ELSIF ref.driveTripOK THEN
    IF ref.driveRelease THEN
        driveStatus.color.fg := COLORS.BLACK;
        driveStatus.color.bg := COLORS.GREEN;
        IF ref.driveMinFrequency THEN
            _formatString(sFormat := '%.1f Hz',  arg1 := F_LREAL(ref.frequencyMeasurement.average.hertz.value), sOut => driveStatus.text);
        ELSE
            _formatString(sFormat := '%.1f Hz (LOW)',  arg1 := F_LREAL(ref.frequencyMeasurement.average.hertz.value), sOut => driveStatus.text);
		END_IF
    ELSE
        driveStatus.color.fg := COLORS.BLACK;
        driveStatus.color.bg := COLORS.GRAY;
        driveStatus.text := 'Not released';
	END_IF
ELSE
        driveStatus.color.fg := COLORS.WHITE;
        driveStatus.color.bg := COLORS.RED;
        driveStatus.text := 'TRIPPED';
END_IF

// update the pressureStatus
pressureStatus(color := HealthToColor(ref.pressureMeasurement.statuses.healthStatus));
_formatString(sFormat := '%.1f Bar',  arg1 := F_LREAL(ref.pressureMeasurement.average.bar.value), sOut => pressureStatus.text);

END_FUNCTION_BLOCK

// ---- MTCS/Hydraulics/Widgets/HydraulicsIOWidget.TcPOU
FUNCTION_BLOCK HydraulicsIOWidget
VAR_INPUT
END_VAR
VAR_OUTPUT
END_VAR
VAR
	actualStatus : StatusWidget;
	pumpsGroup : HydraulicsPumpsGroupIOWidget;
    hydraulicsAndSafety : SafetyHydraulicsAndSafetyIOWidget;
END_VAR
VAR_IN_OUT
	ref : HydraulicsIO;
	ref_safetyIO : SafetyIO;
END_VAR

actualStatus(text  := ref.actualStatus,
             color := HealthToColor(ref.statuses.healthStatus));

pumpsGroup(ref := ref.parts.pumpsGroup);
hydraulicsAndSafety(ref := ref_safetyIO.parts.hydraulicsAndSafety);

END_FUNCTION_BLOCK

// ---- MTCS/Hydraulics/Widgets/HydraulicsPumpsGroupIOWidget.TcPOU
FUNCTION_BLOCK HydraulicsPumpsGroupIOWidget
VAR_INPUT
END_VAR
VAR_OUTPUT
END_VAR
VAR
	actualStatus : StatusWidget;
    
	COU : EtherCatDeviceWidget;
	DI1 : EtherCatDeviceWidget;
	SI1 : EtherCatDeviceWidget;
	SI2 : EtherCatDeviceWidget;
	SI3 : EtherCatDeviceWidget;
	DI2 : EtherCatDeviceWidget;
END_VAR
VAR_IN_OUT
	ref : HydraulicsPumpsGroupIO;
END_VAR

actualStatus(text  := ref.actualStatus,
             color := HealthToColor(ref.statuses.healthStatus));

COU(device := ref.parts.COU);
DI1(device := ref.parts.DI1);
SI1(device := ref.parts.SI1);
SI2(device := ref.parts.SI2);
SI3(device := ref.parts.SI3);
DI2(device := ref.parts.DI2);

END_FUNCTION_BLOCK

// ---- MTCS/Hydraulics/Widgets/HydraulicsWidget.TcPOU
FUNCTION_BLOCK HydraulicsWidget
VAR_INPUT
END_VAR
VAR_OUTPUT
    configManager : ConfigManagerWidget;
	initializationStatus : InitializationStatusWidget;
	actualStatus : StatusWidget;
	pumpsStatus : StatusWidget;
    name : STRING := 'Hydraulics';
    
END_VAR
VAR_IN_OUT
	ref : Hydraulics;
    ref_safetyIO : SafetyIO;
END_VAR
VAR
    io : HydraulicsIOWidget;
    
    button_initialize : InitializeButtonWidget;
    button_operating  : OperatingButtonWidget;
    button_locking    : LockingButtonWidget;
    
    activeTab       : HydraulicsTabs := HydraulicsTabs.OVERVIEW;
    button_overview : SubSystemButtonWidget('Overview'      , HydraulicsTabs.OVERVIEW);
    button_technical: SubSystemButtonWidget('Technical'     , HydraulicsTabs.TECHNICAL);
    button_io       : SubSystemButtonWidget('I/O'           , HydraulicsTabs.IO);
    button_config   : SubSystemButtonWidget('Config'        , HydraulicsTabs.CONFIG);
    
    top             : HydraulicsSideWidget;
    bottom          : HydraulicsSideWidget;
    
	bearingTemperatureStatus : StatusWidget;
    
    _formatString : FB_FormatString;
    activeConfigTab : INT;
    
    bearingTemperature  : MeasurementWidget('Bearing temperature', '%.2f °C');
    topFrequencyMeasurement  : MeasurementWidget('Top drive output frequency', '%.2f Hz');
    topPressureMeasurement  : MeasurementWidget('Top pressure', '%.2f Bar');
    bottomFrequencyMeasurement  : MeasurementWidget('Bottom drive output frequency', '%.2f Hz');
    bottomPressureMeasurement  : MeasurementWidget('Bottom pressure', '%.2f Bar');
    
    circulationStatus : StatusWidget;
    circulationPumpRelay : SimpleRelayWidget;
    pumpsPowerRelay : SimpleRelayWidget;
END_VAR

initializationStatus(status := ref.statuses.initializationStatus);
configManager(mgr := ref.parts.configManager);

actualStatus(text  := ref.actualStatus,
             color := SystemToColor(healthStatus := ref.statuses.healthStatus,
                                    busyStatus   := ref.statuses.busyStatus,
                                    initializationStatus := ref.statuses.initializationStatus,
                                    operatingStatus := ref.statuses.operatingStatus));

pumpsStatus(text  := ref.pumpsStatus, color := actualStatus.color);
                                    
io(ref := ref.parts.io, ref_safetyIO := ref_safetyIO);

button_initialize(status := ref.statuses.initializationStatus, process := ref.processes.initialize);
button_operating(status := ref.statuses.operatingStatus, process := ref.processes.changeOperatingState);
button_locking(status := ref.statuses.initializationStatus, lock := ref.processes.lock, unlock := ref.processes.unlock);

button_overview(    color := actualStatus.color                 , activeTab := activeTab);
button_technical(   color := actualStatus.color                 , activeTab := activeTab);
button_io(          color := io.actualStatus.color              , activeTab := activeTab);
button_config(      color := configManager.actualStatus.color   , activeTab := activeTab);

top(ref := ref.parts.top, powered := ref.parts.pumpsPowerRelay.digitalOutput);
bottom(ref := ref.parts.bottom, powered := ref.parts.pumpsPowerRelay.digitalOutput);

bearingTemperatureStatus(color := HealthToColor(ref.bearingTemperature.statuses.healthStatus));
_formatString(sFormat := '%.1f °C',  arg1 := F_LREAL(ref.bearingTemperature.average.celsius.value), sOut => bearingTemperatureStatus.text);


bearingTemperature(value        := ref.bearingTemperature.average.celsius.value, 
                   actualStatus := ref.bearingTemperature.actualStatus, 
                   healthStatus := ref.bearingTemperature.statuses.healthStatus);
topFrequencyMeasurement(value        := ref.parts.top.frequencyMeasurement.average.hertz.value, 
                        actualStatus := ref.parts.top.frequencyMeasurement.actualStatus, 
                        healthStatus := ref.parts.top.frequencyMeasurement.statuses.healthStatus);
bottomFrequencyMeasurement( value        := ref.parts.bottom.frequencyMeasurement.average.hertz.value, 
                            actualStatus := ref.parts.bottom.frequencyMeasurement.actualStatus, 
                            healthStatus := ref.parts.bottom.frequencyMeasurement.statuses.healthStatus);
topPressureMeasurement(value        := ref.parts.top.pressureMeasurement.average.bar.value, 
                        actualStatus := ref.parts.top.pressureMeasurement.actualStatus, 
                        healthStatus := ref.parts.top.pressureMeasurement.statuses.healthStatus);
bottomPressureMeasurement(value        := ref.parts.bottom.pressureMeasurement.average.bar.value, 
                          actualStatus := ref.parts.bottom.pressureMeasurement.actualStatus, 
                          healthStatus := ref.parts.bottom.pressureMeasurement.statuses.healthStatus);

IF ref.parts.circulationPumpRelay.digitalOutput THEN
    circulationStatus.text := 'ON';
    circulationStatus.color.fg := Colors.BLACK;
    circulationStatus.color.bg := Colors.GREEN;
ELSE
    circulationStatus.text := 'OFF';
    circulationStatus.color.fg := Colors.BLACK;
    circulationStatus.color.bg := Colors.GRAY;
END_IF

circulationPumpRelay(ref := ref.parts.circulationPumpRelay);
pumpsPowerRelay(ref := ref.parts.pumpsPowerRelay);

END_FUNCTION_BLOCK

// ---- MTCS/M1/StateMachines/M1AxialSupport.TcPOU
FUNCTION_BLOCK M1AxialSupport EXTENDS SM_M1AxialSupport
VAR_INPUT
END_VAR
VAR_OUTPUT
END_VAR
VAR
    _unlimitedAutoForceSetpointDaN : LREAL;
    
	_executeController : BOOL;
    _ctrl_pi : FB_CTRL_PI;
    _params  : ST_CTRL_PI_PARAMS;
    
    rawValueSum : LREAL;
    rawValueCount : INT;
    rawValueAverage : DINT;
    
END_VAR

_update();

// calculate the average force
rawValueSum := 0.0;
rawValueCount := 0;
IF (NOT mirrorSouthForce.statuses.healthStatus.bad) AND mirrorSouthForce.statuses.enabledStatus.enabled THEN
    rawValueSum := rawValueSum + DINT_TO_LREAL(mirrorSouthForce.rawValue);
    rawValueCount := rawValueCount + 1;
END_IF
IF (NOT mirrorNorthEastForce.statuses.healthStatus.bad) AND mirrorNorthEastForce.statuses.enabledStatus.enabled THEN
    rawValueSum := rawValueSum + DINT_TO_LREAL(mirrorNorthEastForce.rawValue);
    rawValueCount := rawValueCount + 1;
END_IF
IF (NOT mirrorNorthWestForce.statuses.healthStatus.bad) AND mirrorNorthWestForce.statuses.enabledStatus.enabled THEN
    rawValueSum := rawValueSum + DINT_TO_LREAL(mirrorNorthWestForce.rawValue);
    rawValueCount := rawValueCount + 1;
END_IF

// watch for division by zero!
IF rawValueCount = 0 THEN
    rawValueAverage := 0;
ELSE
    rawValueAverage := LREAL_TO_DINT(rawValueSum / rawValueCount);
END_IF

mirrorAverageForce(
    rawValue   := rawValueAverage,
    error      := rawValueCount = 0,
    underrange := FALSE,
    overrange  := FALSE,
    config     := config.mirrorAverageForce);

// apply any method calls ("processes")
_changePressureSetpointState();
_changePressureSetpoint();


// calculate the automatic force setpoint value in daN
_unlimitedAutoForceSetpointDaN :=  390.0 // force applied by mirror in daN
                                      * config.correctionCoefficient // not really needed, normally 1.0
                                      //* SIN(inclinometer.averageElevation.radians.value)
                                      * SIN(ABS(tubeAngle.radians.value))
                                      / 18.0; // number of support pads

// update the controller setpoint
controllerSetpoint(newNewtonValue := _unlimitedAutoForceSetpointDaN * 10.0);

// only call the _ctrl_pi FB once per task cycle (not once every time the M1AxialSupport FB is called)
IF _executeController <> GLOBAL.config.PLC_TASK_FLIP THEN
	_executeController := GLOBAL.config.PLC_TASK_FLIP;
    
    _params.tCtrlCycleTime    := GLOBAL.config.PLC_CTRL_TIME;
    _params.tTaskCycleTime    := GLOBAL.config.PLC_TASK_TIME;
    _params.bARWOnIPartOnly   := FALSE;
    _params.fKp               := config.controllerKp; 
    _params.tTn               := LREAL_TO_TIME(1000 * config.controllerTn); // 1000 for converting sec to msec
    _params.fOutMaxLimit      := config.controllerLimitMax;
    _params.fOutMinLimit      := config.controllerLimitMin;
    
    
    // setpoint and actualValue are swapped for inverted action!
    IF statuses.pressureSetpointStatus.auto THEN
        _ctrl_pi(
            fSetpointValue  := mirrorAverageForce.average.decaNewton.value,
            fActualValue    := _unlimitedAutoForceSetpointDaN,
            fManSyncValue   := 0.0,
            bSync           := FALSE,
            eMode           := E_CTRL_MODE.eCTRL_MODE_ACTIVE,
            bHold           := FALSE,
            stParams        := _params);
    ELSIF statuses.pressureSetpointStatus.manual THEN
        _ctrl_pi(
            fSetpointValue  := mirrorAverageForce.average.decaNewton.value,
            fActualValue    := _unlimitedAutoForceSetpointDaN,
            fManSyncValue   := 0.0,
            bSync           := FALSE,
            eMode           := E_CTRL_MODE.eCTRL_MODE_RESET,
            bHold           := FALSE,
            stParams        := _params);
    END_IF
    
    autoPressureSetpoint(newBarValue := _ctrl_pi.fOut);
END_IF
    
IF statuses.pressureSetpointStatus.auto THEN
    actualPressureSetpoint(newBarValue := autoPressureSetpoint.bar.value);
    // also update the manualPressureSetpoint
    manualPressureSetpoint(newBarValue := autoPressureSetpoint.bar.value);
    actualStatus := 'Automatic setpoint';
ELSIF statuses.pressureSetpointStatus.manual THEN
    actualPressureSetpoint(newBarValue := manualPressureSetpoint.bar.value);
    actualStatus := 'Fixed setpoint';
END_IF

// update the outputm, but be careful about division-by-zero!
IF config.pressureRegulatorRange = 0 THEN
    pressureSetpointOutput := 0;
ELSE
    pressureSetpointOutput := LREAL_TO_INT(
                                MIN(actualPressureSetpoint.bar.value, config.controllerLimitMax) // [0..max] bar
                                / config.pressureRegulatorRange // e.g. 10 bar
                                * EXPT(2,15)); // 15 bits resolution
END_IF

_update();

METHOD _changePressureSetpoint
VAR_INPUT
END_VAR
IF processes.changePressureSetpoint.statuses.busyStatus.busy THEN
	processes.changePressureSetpoint.setStarted();
    manualPressureSetpoint(newBarValue := processes.changePressureSetpoint.get.setpoint);
	processes.changePressureSetpoint.setFinished();
END_IF
END_METHOD

METHOD _update
VAR_INPUT
END_VAR
SUPER^(config 			:= config,
	   inclinometer 	:= inclinometer,
	   operatorStatus 	:= operatorStatus,
	   operatingStatus 	:= operatingStatus,
       tubeAngle        := tubeAngle);
END_METHOD

METHOD _changePressureSetpointState
VAR_INPUT
END_VAR
IF SUPER^.processes.changePressureSetpointState.statuses.busyStatus.busy THEN
	SUPER^.processes.changePressureSetpointState.setStarted();
	SUPER^.statuses.pressureSetpointStatus(state := SUPER^.processes.changePressureSetpointState.get.state);
	SUPER^.processes.changePressureSetpointState.setFinished();
END_IF
END_METHOD

END_FUNCTION_BLOCK

// ---- MTCS/M1/StateMachines/M1Inclinometer.TcPOU
FUNCTION_BLOCK M1Inclinometer EXTENDS SM_M1Inclinometer
VAR_INPUT
END_VAR
VAR_OUTPUT
END_VAR
VAR
    noOfSamples : UINT := 100;
	_executeMovingAverage : BOOL;
    _ctrl_moving_avg : FB_CTRL_MOVING_AVERAGE;
    _params : ST_CTRL_MOVING_AVERAGE_PARAMS;
    _array : ARRAY [1..100] OF LREAL;
    _cosElevation : LREAL;
END_VAR

_update();

_params.nSamplesToFilter  := noOfSamples;
_params.tCtrlCycleTime    := GLOBAL.config.PLC_CTRL_TIME;

// COS(elevation) * 5V = InclinometerOutput
_cosElevation := voltageMeasurement.actual.volt.value / 5.0; 
IF _cosElevation > 1.0 THEN
    _cosElevation := 1.0;
ELSIF _cosElevation < -1.0 THEN
    _cosElevation := -1.0;
END_IF
actualElevation(newDegreesValue := RadToDeg(ACOS(_cosElevation)));

// only call the _ctrl_moving_avg FB once per task cycle (not once every time the xxxMeasurement FB is called)
IF _executeMovingAverage <> GLOBAL.config.PLC_TASK_FLIP THEN
	_executeMovingAverage := GLOBAL.config.PLC_TASK_FLIP;
	_ctrl_moving_avg(
		fIn             := actualElevation.degrees.value,
		fManSyncValue   := 0.0,
		bSync           := FALSE,
		eMode           := E_CTRL_MODE.eCTRL_MODE_ACTIVE,
		bHold           := FALSE,
		stParams        := _params);
END_IF

averageElevation(newDegreesValue := _ctrl_moving_avg.fOut);

_update();

METHOD _update
VAR_INPUT
END_VAR
SUPER^(config := config);
// update the actualStatus
IF voltageMeasurement.overrange THEN
    actualStatus := 'Overrange';
ELSIF voltageMeasurement.underrange THEN
    actualStatus := 'Underrange';
ELSIF voltageMeasurement.error THEN
    actualStatus := 'Error';
ELSIF statuses.healthStatus.good THEN
    actualStatus := 'OK';
ELSIF statuses.healthStatus.warning THEN
    actualStatus := 'Warning';
ELSE
    actualStatus := 'ERROR';
END_IF
END_METHOD

METHOD FB_init : BOOL
VAR_INPUT
	bInitRetains : BOOL; // if TRUE, the retain variables are initialized (warm start / cold start)
	bInCopyCode : BOOL;  // if TRUE, the instance afterwards gets moved into the copy code (online change)
END_VAR
_params.tTaskCycleTime    := GLOBAL.config.PLC_TASK_TIME;
_params.pWorkArray_ADR    := ADR(_array);
_params.nWorkArray_SIZEOF := SIZEOF(_array);
END_METHOD

END_FUNCTION_BLOCK

// ---- MTCS/M1/StateMachines/M1M2IO.TcPOU
FUNCTION_BLOCK M1M2IO EXTENDS SM_M1M2IO
VAR_INPUT
END_VAR
VAR_OUTPUT
END_VAR
VAR
    _testVar_M1M2IO : BOOL;
END_VAR

SUPER^();

END_FUNCTION_BLOCK

// ---- MTCS/M1/StateMachines/M1RadialSupport.TcPOU
FUNCTION_BLOCK M1RadialSupport EXTENDS SM_M1RadialSupport
VAR_INPUT
END_VAR
VAR_OUTPUT
END_VAR
VAR
    _unlimitedAutoPressureSetpointBar : LREAL;
END_VAR

_update();

_changePressureSetpointState();
_changePressureSetpoint();

// calculate the new value in bar
_unlimitedAutoPressureSetpointBar :=  config.correctionCoefficient 
                                      * 1.33 
                                      *  COS(inclinometer.averageElevation.radians.value);

// update the autoPressureSetpoint, and obey the limits
autoPressureSetpoint(newBarValue := LIMIT(config.controllerLimitMin,
                                          _unlimitedAutoPressureSetpointBar,
                                          config.controllerLimitMax));

// use the autoPressureSetpoint if needed
IF parts.vacuumRelay.digitalOutput THEN
    actualPressureSetpoint(newBarValue := 0.0);
    actualStatus := 'Vacuum ON';
ELSIF statuses.pressureSetpointStatus.auto THEN
    actualPressureSetpoint(newBarValue := autoPressureSetpoint.bar.value);
    // also update the manualPressureSetpoint
    manualPressureSetpoint(newBarValue := autoPressureSetpoint.bar.value);
    actualStatus := 'Automatic setpoint';
ELSIF statuses.pressureSetpointStatus.manual THEN
    actualPressureSetpoint(newBarValue := manualPressureSetpoint.bar.value);
    actualStatus := 'Fixed setpoint';
END_IF

// update the outputm, but be careful about division-by-zero!
IF config.pressureRegulatorRange = 0 THEN
    pressureSetpointOutput := 0;
ELSE
    pressureSetpointOutput := LREAL_TO_INT(
                                MIN(actualPressureSetpoint.bar.value, config.controllerLimitMax) // [0..max] bar
                                / config.pressureRegulatorRange // e.g. 10 bar
                                * EXPT(2,15)); // 15 bits resolution
END_IF

// update the statemachine
_update();

METHOD _changePressureSetpoint
VAR_INPUT
END_VAR
IF processes.changePressureSetpoint.statuses.busyStatus.busy THEN
	processes.changePressureSetpoint.setStarted();
    manualPressureSetpoint(newBarValue := processes.changePressureSetpoint.get.setpoint);
	processes.changePressureSetpoint.setFinished();
END_IF
END_METHOD

METHOD _changePressureSetpointState
VAR_INPUT
END_VAR
IF SUPER^.processes.changePressureSetpointState.statuses.busyStatus.busy THEN
	SUPER^.processes.changePressureSetpointState.setStarted();
	SUPER^.statuses.pressureSetpointStatus(state := SUPER^.processes.changePressureSetpointState.get.state);
	SUPER^.processes.changePressureSetpointState.setFinished();
END_IF
END_METHOD

METHOD _update
VAR_INPUT
END_VAR
SUPER^(config 			:= config,
	   inclinometer 	:= inclinometer,
	   operatorStatus 	:= operatorStatus,
	   operatingStatus 	:= operatingStatus);
END_METHOD

END_FUNCTION_BLOCK

// ---- MTCS/M1/Widgets/M1AxialSupportWidget.TcPOU
FUNCTION_BLOCK M1AxialSupportWidget
VAR_INPUT
END_VAR
VAR_OUTPUT
END_VAR
VAR_IN_OUT
    ref : M1AxialSupport;
END_VAR
VAR
	actualStatus  : StatusWidget;
    
    regulatorPressure      : MeasurementWidget('Axial pressure @ regulator'     , '%.2f bar');
    mirrorPressure         : MeasurementWidget('Axial pressure @ mirror cell'   , '%.2f bar');
    mirrorSouthForce       : MeasurementWidget('Axial force @ South (SO)'       , '%.2f daN');
    mirrorNorthEastForce   : MeasurementWidget('Axial force @ North-East (NE)'  , '%.2f daN');
    mirrorNorthWestForce   : MeasurementWidget('Axial force @ North-West (NW)'  , '%.2f daN');
    mirrorAverageForce     : MeasurementWidget('Axial force Average'            , '%.2f daN');
    
    changeToAutoButtonDeactivated : BOOL;
    changeToManualButtonDeactivated : BOOL;
    
    operatingStatus : StatusWidget; 
END_VAR

actualStatus(text  := ref.actualStatus, 
             color := HealthBusyToColor(healthStatus := ref.statuses.healthStatus,
                                        busyStatus   := ref.statuses.busyStatus));

regulatorPressure( value        := ref.regulatorPressure.average.bar.value, 
                   actualStatus := ref.regulatorPressure.actualStatus, 
                   healthStatus := ref.regulatorPressure.statuses.healthStatus);
mirrorPressure( value        := ref.mirrorPressure.average.bar.value, 
                actualStatus := ref.mirrorPressure.actualStatus, 
                healthStatus := ref.mirrorPressure.statuses.healthStatus);
                
mirrorSouthForce( 
    value        := ref.mirrorSouthForce.average.decaNewton.value, 
    actualStatus := ref.mirrorSouthForce.actualStatus, 
    healthStatus := ref.mirrorSouthForce.statuses.healthStatus);
mirrorNorthEastForce( 
    value        := ref.mirrorNorthEastForce.average.decaNewton.value, 
    actualStatus := ref.mirrorNorthEastForce.actualStatus, 
    healthStatus := ref.mirrorNorthEastForce.statuses.healthStatus);
mirrorNorthWestForce( 
    value        := ref.mirrorNorthWestForce.average.decaNewton.value, 
    actualStatus := ref.mirrorNorthWestForce.actualStatus, 
    healthStatus := ref.mirrorNorthWestForce.statuses.healthStatus);
mirrorAverageForce( 
    value        := ref.mirrorAverageForce.average.decaNewton.value, 
    actualStatus := ref.mirrorAverageForce.actualStatus, 
    healthStatus := ref.mirrorAverageForce.statuses.healthStatus);
    
changeToAutoButtonDeactivated := ref.processes.changePressureSetpointState.statuses.enabledStatus.disabled
                                 OR ref.statuses.pressureSetpointStatus.auto;
changeToManualButtonDeactivated := ref.processes.changePressureSetpointState.statuses.enabledStatus.disabled
                                   OR ref.statuses.pressureSetpointStatus.manual;
                                   
IF ref.statuses.pressureSetpointStatus.auto THEN
    operatingStatus(text := 'Automatic');
    operatingStatus.color.bg := Colors.GREEN;
    operatingStatus.color.fg := Colors.WHITE;
ELSIF ref.statuses.pressureSetpointStatus.manual THEN
    operatingStatus(text := 'Fixed');
    operatingStatus.color.bg := Colors.ORANGE;
    operatingStatus.color.fg := Colors.WHITE;
END_IF

END_FUNCTION_BLOCK

// ---- MTCS/M1/Widgets/M1FigureWidget.TcPOU
FUNCTION_BLOCK M1FigureWidget
VAR_INPUT
END_VAR
VAR_OUTPUT
END_VAR
VAR_IN_OUT
    ref : M1;
END_VAR
VAR
    axialSouthAngle : REAL := 0;
    axialNorthEastAngle : REAL := 120;
    axialNorthWestAngle : REAL := 240;
    
    radPad0Angle : REAL := -30-1*(120/5);
    radPad1Angle : REAL := -30-2*(120/5);
    radPad2Angle : REAL := -30-3*(120/5);
    radPad3Angle : REAL := -30-4*(120/5);
    
    axPad0Angle : REAL := 1* 30;
    axPad1Angle : REAL := 2* 30;
    axPad2Angle : REAL := 3* 30;
    axPad3Angle : REAL := 5* 30;
    axPad4Angle : REAL := 6* 30;
    axPad5Angle : REAL := 7* 30;
    axPad6Angle : REAL := 9* 30;
    axPad7Angle : REAL := 10* 30;
    axPad8Angle : REAL := 11* 30;
    
    axPadInner0Angle : LREAL := -15 + 0*60;
    axPadInner1Angle : LREAL := -15 + 1*60;
    axPadInner2Angle : LREAL := -15 + 2*60;
    axPadInner3Angle : LREAL := -15 + 3*60;
    axPadInner4Angle : LREAL := -15 + 4*60;
    axPadInner5Angle : LREAL := -15 + 5*60;
    
    supplyPressureString : STRING;
    axialRegulatorPressureString : STRING;
    axialMirrorPressureString : STRING;
    axialRegulatorSetpointString : STRING;
    radialRegulatorPressureString : STRING;
    radialMirrorPressureString : STRING;
    radialRegulatorSetpointString : STRING;
    axialForceStringSO : STRING;
    axialForceStringNE : STRING;
    axialForceStringNW : STRING;
    
    _formatString : FB_FormatString;
END_VAR

supplyPressureString            := _getPressureMeasurementString(ref.pneumaticSupplyPressure);
radialRegulatorPressureString   := _getPressureMeasurementString(ref.parts.radialSupport.regulatorPressure);
radialMirrorPressureString      := _getPressureMeasurementString(ref.parts.radialSupport.mirrorPressure);
radialRegulatorSetpointString   := _getPressureSetpointString(ref.parts.radialSupport.actualPressureSetpoint);
axialRegulatorPressureString    := _getPressureMeasurementString(ref.parts.axialSupport.regulatorPressure);
axialMirrorPressureString       := _getPressureMeasurementString(ref.parts.axialSupport.mirrorPressure);
axialRegulatorSetpointString    := _getPressureSetpointString(ref.parts.axialSupport.actualPressureSetpoint);
axialForceStringSO              := _getForceMeasurementString(ref.parts.axialSupport.mirrorSouthForce);
axialForceStringNE              := _getForceMeasurementString(ref.parts.axialSupport.mirrorNorthEastForce);
axialForceStringNW              := _getForceMeasurementString(ref.parts.axialSupport.mirrorNorthWestForce);

METHOD _getPressureMeasurementString : STRING
VAR_INPUT
END_VAR
VAR_IN_OUT
    measurement : PressureMeasurement;
END_VAR
_getPressureMeasurementString := _getValueString(
        value           := measurement.average.bar.value,
        format          := '%.1f bar',
        underrange      := measurement.underrange,
        overrange       := measurement.overrange,
        error           := measurement.error,
        enabled         := measurement.statuses.enabledStatus.enabled,
        disabled        := measurement.statuses.enabledStatus.disabled);
END_METHOD

METHOD _getPressureSetpointString : STRING
VAR_INPUT
END_VAR
VAR_IN_OUT
    setpoint : Pressure;
END_VAR
_formatString(sFormat := '%.1f bar', 
              arg1    := F_LREAL(setpoint.bar.value),
              sOut    => _getPressureSetpointString);
END_METHOD

METHOD _getValueString : STRING
VAR_INPUT
    value : LREAL;
    format : STRING;
    underrange : BOOL;
    overrange : BOOL;
    error : BOOL;
    enabled : BOOL;
    disabled : BOOL;
END_VAR
IF disabled THEN
    _getValueString := 'Disabled';
ELSIF enabled THEN
    IF underrange THEN
        _getValueString := 'Underrange';
    ELSIF overrange THEN
        _getValueString := 'Overrange';
    ELSIF error THEN
        _getValueString := 'Error';
    ELSE
        _formatString(sFormat := format, 
                      arg1    := F_LREAL(value),
                      sOut    => _getValueString);
	END_IF
ELSE
    _getValueString := '';
END_IF
END_METHOD

METHOD _getForceMeasurementString : STRING
VAR_INPUT
END_VAR
VAR_IN_OUT
    measurement : ForceMeasurement;
END_VAR
_getForceMeasurementString := _getValueString(
        value           := measurement.average.decaNewton.value,
        format          := '%.1f daN',
        underrange      := measurement.underrange,
        overrange       := measurement.overrange,
        error           := measurement.error,
        enabled         := measurement.statuses.enabledStatus.enabled,
        disabled        := measurement.statuses.enabledStatus.disabled);
END_METHOD

END_FUNCTION_BLOCK

// ---- MTCS/M1/Widgets/M1RadialSupportWidget.TcPOU
FUNCTION_BLOCK M1RadialSupportWidget
VAR_INPUT
END_VAR
VAR_OUTPUT
END_VAR
VAR_IN_OUT
    ref : M1RadialSupport;
END_VAR
VAR
	actualStatus  : StatusWidget;
    
    regulatorPressure : MeasurementWidget('Radial pressure @ regulator', '%.2f bar');
    mirrorPressure : MeasurementWidget('Radial pressure @ mirror cell' , '%.2f bar');
    
    changeToAutoButtonDeactivated : BOOL;
    changeToManualButtonDeactivated : BOOL;
    
    operatingStatus : StatusWidget; 
    
    vacuumRelay : SimpleRelayWidget;
END_VAR

actualStatus(text  := ref.actualStatus, 
             color := HealthBusyToColor(healthStatus := ref.statuses.healthStatus,
                                        busyStatus   := ref.statuses.busyStatus));

regulatorPressure( value        := ref.regulatorPressure.average.bar.value, 
                   actualStatus := ref.regulatorPressure.actualStatus, 
                   healthStatus := ref.regulatorPressure.statuses.healthStatus);
mirrorPressure( value        := ref.mirrorPressure.average.bar.value, 
                actualStatus := ref.mirrorPressure.actualStatus, 
                healthStatus := ref.mirrorPressure.statuses.healthStatus);
                
changeToAutoButtonDeactivated := ref.processes.changePressureSetpointState.statuses.enabledStatus.disabled
                                 OR ref.statuses.pressureSetpointStatus.auto;
changeToManualButtonDeactivated := ref.processes.changePressureSetpointState.statuses.enabledStatus.disabled
                                   OR ref.statuses.pressureSetpointStatus.manual;
                                   
IF ref.statuses.pressureSetpointStatus.auto THEN
    operatingStatus(text := 'Automatic');
    operatingStatus.color.bg := Colors.GREEN;
    operatingStatus.color.fg := Colors.WHITE;
ELSIF ref.statuses.pressureSetpointStatus.manual THEN
    operatingStatus(text := 'Fixed');
    operatingStatus.color.bg := Colors.ORANGE;
    operatingStatus.color.fg := Colors.WHITE;
END_IF

vacuumRelay(ref := ref.parts.vacuumRelay);

END_FUNCTION_BLOCK

// ---- MTCS/M1/Widgets/M1M2IOWidget.TcPOU
FUNCTION_BLOCK M1M2IOWidget
VAR_INPUT
END_VAR
VAR_OUTPUT
END_VAR
VAR
	actualStatus : StatusWidget;
    COU  : EtherCatDeviceWidget;
    AI1  : EtherCatDeviceWidget;
    AI2  : EtherCatDeviceWidget;
    AI3  : EtherCatDeviceWidget;
    AO1  : EtherCatDeviceWidget;
    DO1  : EtherCatDeviceWidget;
    RES1   : EtherCatDeviceWidget;
    RES2   : EtherCatDeviceWidget;
    RES3   : EtherCatDeviceWidget;
    PWR1   : EtherCatDeviceWidget;
    SSI1   : EtherCatDeviceWidget;
    AI4  : EtherCatDeviceWidget;
    INC1   : EtherCatDeviceWidget;
    P5V1   : EtherCatDeviceWidget;
    DO2  : EtherCatDeviceWidget;
    DO3    : EtherCatDeviceWidget;
    RE1    : EtherCatDeviceWidget;
END_VAR
VAR_IN_OUT
	ref : M1M2IO;
END_VAR

actualStatus(text  := ref.actualStatus,
             color := HealthToColor(ref.statuses.healthStatus));

COU(device := ref.parts.COU);
AI1(device := ref.parts.AI1);
AI2(device := ref.parts.AI2);
AI3(device := ref.parts.AI3);
AO1(device := ref.parts.AO1);
DO1(device := ref.parts.DO1);
RES1(device := ref.parts.RES1);
RES2(device := ref.parts.RES2);
RES3(device := ref.parts.RES3);
PWR1(device := ref.parts.PWR1);
SSI1(device := ref.parts.SSI1);
AI4(device := ref.parts.AI4);
INC1(device := ref.parts.INC1);
P5V1(device := ref.parts.P5V1);
DO2(device := ref.parts.DO2);
DO3(device := ref.parts.DO3);
RE1(device := ref.parts.RE1);

END_FUNCTION_BLOCK

// ---- MTCS/M1/Widgets/M1InclinometerWidget.TcPOU
FUNCTION_BLOCK M1InclinometerWidget
VAR_INPUT
END_VAR
VAR_OUTPUT
END_VAR
VAR_IN_OUT
    ref : M1Inclinometer;
END_VAR
VAR
	actualStatus        : StatusWidget;
    voltageMeasurement  : MeasurementWidget('Inclinometer voltage', '%.2f V');
    elevation           : MeasurementWidget('Inclinometer angle (not used)', '%.2f °');
END_VAR

actualStatus(text  := ref.actualStatus, 
             color := HealthToColor(healthStatus := ref.voltageMeasurement.statuses.healthStatus));

voltageMeasurement( 
    value        := ref.voltageMeasurement.average.volt.value, 
    actualStatus := ref.voltageMeasurement.actualStatus, 
    healthStatus := ref.voltageMeasurement.statuses.healthStatus);
    
elevation(
    value        := ref.averageElevation.degrees.value,
    actualStatus := ref.actualStatus, 
    healthStatus := ref.statuses.healthStatus);

END_FUNCTION_BLOCK

// ---- MTCS/M1/Widgets/M1Widget.TcPOU
FUNCTION_BLOCK M1Widget
VAR_INPUT
    activeTab : M1Tabs := M1Tabs.OVERVIEW;
END_VAR
VAR_OUTPUT
    name : STRING := 'M1';
END_VAR
VAR_IN_OUT
	ref : M1;
    ref_tubeAngleMeasurement : TelemetryAccelerometer;
END_VAR
VAR
	actualStatus            : StatusWidget;
	initializationStatus    : InitializationStatusWidget;
	
    button_initialize 	: InitializeButtonWidget;
    button_operating  	: OperatingButtonWidget;
    button_locking    	: LockingButtonWidget;
    
    button_overview   	: SubSystemButtonWidget('Overview'		, M1Tabs.OVERVIEW);
    button_radial     	: SubSystemButtonWidget('Radial' 	    , M1Tabs.RADIAL);
    button_axial      	: SubSystemButtonWidget('Axial' 	    , M1Tabs.AXIAL);
    button_io         	: SubSystemButtonWidget('I/O'    		, M1Tabs.IO);
    button_config     	: SubSystemButtonWidget('Config'  		, M1Tabs.CONFIG);
    
    radialSupport       : M1RadialSupportWidget;
    axialSupport        : M1AxialSupportWidget;
    inclinometer        : M1InclinometerWidget;
    io 					: M1M2IOWidget;
    configManager       : ConfigManagerWidget;
    
    figure              : M1FigureWidget;
    
    activeConfigTab : INT;
    
    pneumaticSupplyPressure   : MeasurementWidget('Pneumatic supply pressure', '%.2f bar');
    
    accelerometerAngle : MeasurementWidget('Accelerometers angle (used!)', '%.2f °');
END_VAR

initializationStatus(status := ref.statuses.initializationStatus);


button_initialize(status := ref.statuses.initializationStatus, process := ref.processes.initialize);
button_operating(status := ref.statuses.operatingStatus, process := ref.processes.changeOperatingState);
button_locking(status := ref.statuses.initializationStatus, lock := ref.processes.lock, unlock := ref.processes.unlock);

button_overview(    color := actualStatus.color                 , activeTab := activeTab);
button_radial(      color := radialSupport.actualStatus.color   , activeTab := activeTab);
button_axial(       color := axialSupport.actualStatus.color   	, activeTab := activeTab);
button_io(          color := io.actualStatus.color              , activeTab := activeTab);
button_config(      color := configManager.actualStatus.color   , activeTab := activeTab);

radialSupport(ref := ref.parts.radialSupport);
axialSupport(ref := ref.parts.axialSupport);
inclinometer(ref := ref.parts.inclinometer);
io(ref := ref.parts.io);
configManager(mgr := ref.parts.configManager);

figure(ref := ref);

actualStatus(text  := ref.actualStatus,
             color := SystemToColor(healthStatus := ref.statuses.healthStatus,
                                    busyStatus   := ref.statuses.busyStatus,
                                    initializationStatus := ref.statuses.initializationStatus,
                                    operatingStatus := ref.statuses.operatingStatus));

pneumaticSupplyPressure( 
    value        := ref.pneumaticSupplyPressure.average.bar.value, 
    actualStatus := ref.pneumaticSupplyPressure.actualStatus, 
    healthStatus := ref.pneumaticSupplyPressure.statuses.healthStatus);
    
accelerometerAngle(
    value        := ABS(ref_tubeAngleMeasurement.averageYAngle.degrees.value),  // ABS !!!
    actualStatus := ref_tubeAngleMeasurement.actualStatus, 
    healthStatus := ref_tubeAngleMeasurement.statuses.yHealthStatus);

END_FUNCTION_BLOCK

// ---- MTCS/M2/Helper/M2AxisToAddress.TcPOU
FUNCTION M2AxisToAddress : WORD
VAR_INPUT
    axis : M2Axes;
END_VAR
VAR
END_VAR

CASE axis OF                   // ABC
    M2Axes.Z:
        M2AxisToAddress := 0;  // 000
    M2Axes.Y:
        M2AxisToAddress := 1;  // 100
    M2Axes.X:
        M2AxisToAddress := 2;  // 010
    M2Axes.TILTY:
        M2AxisToAddress := 3;  // 110
    M2Axes.TILTX:
        M2AxisToAddress := 4;  // 001
END_CASE

END_FUNCTION

// ---- MTCS/M2/Helper/M2AddressToAxis.TcPOU
FUNCTION M2AddressToAxis : M2Axes
VAR_INPUT
    address : WORD;
END_VAR
VAR
END_VAR

CASE address OF
    0:
        M2AddressToAxis := M2Axes.Z;
    1:
        M2AddressToAxis := M2Axes.Y;
    2:
        M2AddressToAxis := M2Axes.X;
    3:
        M2AddressToAxis := M2Axes.TILTY;
    4:
        M2AddressToAxis := M2Axes.TILTX;
END_CASE

END_FUNCTION

// ---- MTCS/M2/Helper/M2AxisToGeneralConfig.TcPOU
FUNCTION M2AxisToGeneralConfig : M2AxisGeneralConfig
VAR_INPUT
    axis : M2Axes;
END_VAR
VAR_IN_OUT
    config : M2Config;
END_VAR
VAR
END_VAR

CASE axis OF
    M2Axes.X:
        M2AxisToGeneralConfig := config.x.general;
    M2Axes.Y:
        M2AxisToGeneralConfig := config.y.general;
    M2Axes.Z:
        M2AxisToGeneralConfig := config.z.general;
    M2Axes.TILTX:
        M2AxisToGeneralConfig := config.tiltX.general;
    M2Axes.TILTY:
        M2AxisToGeneralConfig := config.tiltY.general;
END_CASE

END_FUNCTION

// ---- MTCS/M2/Helper/M2AxisToString.TcPOU
FUNCTION M2AxisToString : STRING
VAR_INPUT
    axis : M2Axes;
END_VAR
VAR
END_VAR

CASE axis OF
    M2Axes.Z:
        M2AxisToString := 'Z';
    M2Axes.Y:
        M2AxisToString := 'Y';
    M2Axes.X:
        M2AxisToString := 'X';
    M2Axes.TILTY:
        M2AxisToString := 'Tilt Y';
    M2Axes.TILTX:
        M2AxisToString := 'Tilt X';
END_CASE

END_FUNCTION

// ---- MTCS/M2/Helper/M2ComputeAbsoluteMove.TcPOU
FUNCTION M2ComputeAbsoluteMove : BOOL
VAR_INPUT
    initialPosition : LREAL;
    finalPosition : LREAL;
    gearReduction : LREAL;
    feedbackResolution : LREAL;
    screwPitch : LREAL;
END_VAR
VAR_OUTPUT
    steps : UDINT;
    cw : BOOL;
    deltaPosition : LREAL;
END_VAR
VAR
END_VAR

// first calculate the delta position in micrometers
deltaPosition := finalPosition - initialPosition;

// the CCW or CW sense depends on the sign of the delta
cw := (deltaPosition < 0);

// calculate the steps (LREAL_TO_UDINT rounds the number instead of truncating it!)
steps := LREAL_TO_UDINT( ABS(deltaPosition) * gearReduction * feedbackResolution / screwPitch );

END_FUNCTION

// ---- MTCS/M2/Helper/M2ComputeThermalFocusFromId.TcPOU
FUNCTION M2ComputeThermalFocusFromId : LREAL // returns position in mm
VAR_INPUT
    positionId : M3PositionIDs;
END_VAR
VAR_IN_OUT
    config : M2ThermalFocusConfig;
    temperatures : TelemetryTemperatures;
END_VAR
VAR
END_VAR


CASE positionId OF
    M3PositionIDs.CASSEGRAIN:
        M2ComputeThermalFocusFromId := M2ComputeThermalFocus(config := config.cassegrain, temperatures);
    M3PositionIDs.NASMYTH_A:
        M2ComputeThermalFocusFromId := M2ComputeThermalFocus(config := config.nasmythA, temperatures);
    M3PositionIDs.NASMYTH_B:
        M2ComputeThermalFocusFromId := M2ComputeThermalFocus(config := config.nasmythB, temperatures);
    M3PositionIDs.NASMYTH_C:
        M2ComputeThermalFocusFromId := M2ComputeThermalFocus(config := config.nasmythC, temperatures);
    M3PositionIDs.NASMYTH_D:
        M2ComputeThermalFocusFromId := M2ComputeThermalFocus(config := config.nasmythD, temperatures);
    M3PositionIDs.OTHER_0:
        M2ComputeThermalFocusFromId := M2ComputeThermalFocus(config := config.other0, temperatures);
    M3PositionIDs.OTHER_1:
        M2ComputeThermalFocusFromId := M2ComputeThermalFocus(config := config.other1, temperatures);
    M3PositionIDs.OTHER_2:
        M2ComputeThermalFocusFromId := M2ComputeThermalFocus(config := config.other2, temperatures);
    M3PositionIDs.OTHER_3:
        M2ComputeThermalFocusFromId := M2ComputeThermalFocus(config := config.other3, temperatures);
    M3PositionIDs.OTHER_4:
        M2ComputeThermalFocusFromId := M2ComputeThermalFocus(config := config.other4, temperatures);
    M3PositionIDs.UNKNOWN:
        M2ComputeThermalFocusFromId := 0.0;
END_CASE

END_FUNCTION

// ---- MTCS/M2/Helper/M2ComputeThermalFocus.TcPOU
FUNCTION M2ComputeThermalFocus : LREAL // returns position in mm
VAR_INPUT
END_VAR
VAR_IN_OUT
    config : M2ThermalFocusStationConfig;
    temperatures : TelemetryTemperatures;
END_VAR
VAR
END_VAR

M2ComputeThermalFocus := config.offset
                         + config.topCoefficient * temperatures.topTube.average.celsius.value
                         + config.centreCoefficient * temperatures.centreTube.average.celsius.value
                         + config.mirrorCellCoefficient * temperatures.mirrorCell.average.celsius.value;

END_FUNCTION

// ---- MTCS/M2/StateMachines/M2TiltXAxis.TcPOU
FUNCTION_BLOCK M2TiltXAxis EXTENDS SM_M2TiltXAxis
VAR_INPUT
END_VAR
VAR_OUTPUT
END_VAR
VAR
    _lastRawValue : INT;
END_VAR


IF powered THEN
    _lastRawValue := SUPER^.position.rawValue;
ELSE
   SUPER^.position.rawValue := _lastRawValue;
END_IF

statuses.healthStatus(isGood := TRUE);

SUPER^(config := SUPER^.config, axisConfig := SUPER^.axisConfig);

END_FUNCTION_BLOCK

// ---- GlobalTextList.TcGTLO
TEXTLIST GlobalTextList
  29 = '\nObserver'
  798 = '\nOFF\ndelay\n4 sec'
  28 = '\nTech'
  231 = '                average current'
  1564 = '  0°\nN'
  1010 = ' - coefficient a'
  1011 = ' - coefficient b'
  1012 = ' - coefficient c'
  1563 = ' 0°\nN'
  1991 = ' 8s'
  1644 = ' <<< Move out <<<'
  1931 = ' step'
  208 = ' T'
  668 = '!'
  968 = '!!! Only do this in case you cannot recover the system in another way !!!'
  1771 = '"'
  1242 = '"Person has left" button is pressed'
  1241 = '"Person has left" button is pushed'
  506 = '$s'
  556 = '%,3f'
  1855 = '%.01f"'
  1514 = '%.02f'
  1518 = '%.02f"'
  1519 = '%.02f" '
  1767 = '%.0f'
  1867 = '%.1'
  1868 = '%.1 '
  1865 = '%.1 " /s'
  1866 = '%.1 arcsec / s'
  41 = '%.1f'
  1787 = '%.1f "/s'
  1788 = '%.1f "/s²'
  1508 = '%.1f %'
  986 = '%.1f Hz'
  411 = '%.1f m'
  1524 = '%.1f Nm'
  417 = '%.1f °'
  473 = '%.1f °/s'
  1939 = '%.1f"'
  1790 = '%.1f"/s'
  63 = '%.2f'
  652 = '%.2f daN'
  653 = '%.2f daN '
  1739 = '%.2f °/s'
  223 = '%.3f'
  1789 = '%.3f "/s²'
  1507 = '%.3f %'
  1496 = '%.3f A'
  557 = '%.3f bar'
  1306 = '%.3f mm'
  1501 = '%.3f Nm'
  1527 = '%.3f Nm (motor)'
  1504 = '%.3f Nm/A'
  1796 = '%.3f °/s'
  1791 = '%.3f"/s²'
  1060 = '%.4 mm'
  18 = '%.4f'
  84 = '%.4f '
  158 = '%.4f %s'
  541 = '%.4f bar'
  651 = '%.4f daN'
  72 = '%.4f mm'
  1944 = '%.4f mm/s'
  12 = '%.4f °'
  472 = '%.4f °/s'
  77 = '%.4f°'
  2103 = '%.4f°/s'
  1387 = '%.5f'
  1388 = '%.6f'
  360 = '%.8f'
  1116 = '%.f mG'
  505 = '%.s'
  386 = '%1d'
  387 = '%2d'
  385 = '%3d'
  9 = '%d'
  1105 = '%d '
  1786 = '%d "/s'
  454 = '%d mA'
  1107 = '%d mG'
  419 = '%d °'
  1785 = '%d" /s'
  420 = '%df °'
  5 = '%s'
  515 = '%s  '
  2113 = '%s %.0f°'
  1431 = '%s ...'
  1392 = '%s / s'
  1393 = '%s / s2'
  1394 = '%s / s²'
  1402 = '%s /s'
  1403 = '%s /s²'
  335 = "%s'"
  293 = '%x'
  1770 = "'"
  1218 = '(0 = repeat pattern forever)'
  1217 = '(0 means: repeat pattern forever)'
  737 = '(at low speed!'
  735 = '(at low speed!)'
  283 = '(b)'
  292 = '(dec)'
  1380 = '(e.g. 2000.0)'
  291 = '(hex)'
  734 = '(low speed!)'
  1205 = '(NOT recommended'
  1207 = '(Not recommended!)'
  510 = '+'
  1928 = '+ a'
  1742 = '+ AZI'
  1886 = '+ Azimuth'
  721 = '+ c * centreTemperature'
  1893 = '+ Cassegrain\nrotation'
  719 = '+ centre * centreTemperature'
  715 = '+ centre * centreTemperature + mirrorCell * mirrorCellTemperature'
  1926 = '+ d'
  1740 = '+ ELE'
  1884 = '+ Elevation'
  722 = '+ m * mirrorCellTemperature'
  718 = '+ mirrorCell * mirrorCellTemperature'
  1895 = '+ Nasmyth\nrotation'
  1799 = '+ ROC'
  1956 = '+ RON'
  1954 = '+ ROT'
  1905 = '+ Rotation'
  720 = '+ t * topTemperature'
  716 = '+ top * topTemperature'
  713 = '+ top * topTemperature + centre * centreTemperature + mirrorCell * mirrorCellTemperature'
  1747 = '+34* 52\' 44.8"'
  692 = '+tilt X'
  693 = '+tiltX'
  698 = '+tiltY'
  690 = '+X'
  1101 = '+X1'
  695 = '+Y'
  1103 = '+Y1'
  1114 = '+Y2'
  699 = '+Z'
  85 = '-'
  1903 = '-\nAzimuth'
  1930 = '- a'
  1743 = '- AZI'
  1887 = '- Azimuth'
  281 = '- bin'
  1892 = '- Cassegrain\nrotation'
  1927 = '- d'
  279 = '- dec'
  1741 = '- ELE'
  1885 = '- Elevation'
  280 = '- hex'
  1894 = '- Nasmyth\nrotation'
  1798 = '- ROC'
  1955 = '- RON'
  1797 = '- ROT'
  1904 = '- Rotation'
  1817 = '-300* 55\' 55"'
  1818 = '-300* 55\' 55.5"'
  1823 = '-300* 55\' 55.5"\n-300.2423*'
  1822 = '-300* 55\' 55.5"\n-300.242342'
  1819 = '-300* 55\' 55.5" (-300.8750)'
  1820 = '-300* 55\' 55.5" (-300.8750*)'
  1821 = '-300* 55\' 55.5" = -300.8750*)'
  1779 = '-334* 52\' 44.8"'
  1929 = '-a '
  694 = '-tilt X'
  697 = '-tiltY'
  691 = '-X'
  1113 = '-X2'
  696 = '-Y'
  700 = '-Z'
  1104 = '-Z1'
  1115 = '-Z2'
  44 = '...'
  245 = '... at position'
  1808 = '... for'
  1924 = '/'
  1882 = '/ hour'
  1883 = '/ minute'
  1881 = '/ s'
  149 = '0'
  1726 = '0.1 °/s'
  1732 = '0.10 °/s'
  1795 = '0.1000 °/s'
  2104 = '0.332°/s'
  1794 = '0.3333 °/s'
  282 = '01234567890123456'
  164 = '0x%d'
  163 = '0x%x'
  1552 = '0°'
  1562 = '0°\nN'
  1554 = '0° N'
  103 = '1'
  1725 = '1 °/s'
  614 = '1.3 bar'
  619 = '1.33 daN'
  1727 = '1.5 °/s'
  1733 = '1.50 °/s'
  1749 = '12* 34\' 56.5"'
  1746 = '12h 34m 56.5s'
  167 = '16#%d'
  166 = '16#%x'
  165 = '16%x'
  1553 = '180°'
  1555 = '180° S'
  104 = '2'
  620 = '200.3 daN'
  1062 = '22.2222'
  1059 = '22.2222 mm'
  1556 = '270° E'
  1559 = '270° S'
  1560 = '270° W'
  507 = '2800.0000  + 30'
  143 = '3'
  1724 = '3 °/s'
  1723 = '3 ↑'
  1731 = '3.0 °/s'
  1734 = '3.00 °/s'
  1750 = '356* 34\' 56.5"'
  1753 = '36* 34\' 56.5"'
  105 = '4'
  144 = '5'
  145 = '6'
  1768 = '66'
  1772 = '66.6'
  146 = '7'
  1989 = '7s'
  147 = '8'
  1990 = '8s'
  148 = '9'
  1566 = '90°'
  1557 = '90° (E)'
  1551 = '90° E'
  377 = ':'
  1056 = '<'
  1645 = '<<< Move out <<<'
  1510 = '='
  1966 = '= Sufficiently high?'
  1967 = '= sufficiently high?'
  1503 = '==> Torque constant'
  1057 = '>'
  1295 = '>>>'
  1648 = '>>> Move out'
  1298 = '?'
  806 = '@ control room'
  804 = '@ dome'
  1230 = '@ dome 1'
  1231 = '@ dome 2'
  1232 = '@ dome access'
  805 = '@ first floor'
  1525 = '@ motor'
  1526 = '@ telescope'
  222 = 'A'
  1744 = 'a'
  1935 = 'a & d'
  1934 = 'a + d'
  1186 = 'A person has entered the dome'
  2095 = 'ABL'
  1633 = 'ABL axis'
  228 = 'ABL motor actual current'
  233 = 'ABL motor average current'
  234 = 'ABL motor offset'
  235 = 'ABL motor position'
  1523 = 'ABL motor torque'
  219 = 'Abort'
  1076 = 'ABORT'
  331 = 'Abort\nprocedure'
  332 = 'Abort / reset'
  1600 = 'Absolute'
  1601 = 'Absolute enc.'
  1596 = 'Absolute encoder'
  1718 = 'Absolute encoder position where the homing should go to first, in degrees'
  1680 = 'Acceleration or deceleration of the physical axis, in degrees/sec^2 (>0)'
  1681 = 'Acceleration/deceleration limit of the physical axis, in degrees/sec^2 (>0)'
  1112 = 'Accelerometer angles'
  1111 = 'Accelerometers'
  1992 = 'Access OK'
  1471 = 'ACEC'
  1469 = 'ACES'
  2058 = 'Acknowledge'
  809 = 'Acknowledge error(s)'
  2108 = 'Act position'
  1625 = 'actAcc'
  4 = 'ACTIVATE'
  43 = 'Active'
  2 = 'Active\nconfig'
  1623 = 'actPos'
  1816 = 'ActPos'
  1628 = 'actPos,'
  1629 = 'actPos,\nactVelo,\nactAcc'
  1631 = 'actPos/Vel/Acc'
  1630 = 'actPos/Velo/Acc'
  1815 = 'ActPos:'
  1117 = 'Actual'
  1863 = 'Actual alpha velocity:'
  1023 = 'Actual bottom setpoint:'
  1043 = 'Actual counter value: %d'
  462 = 'Actual current'
  461 = 'Actual current (0-8 panels!):'
  467 = 'Actual current:'
  1864 = 'Actual delta velocity:'
  393 = 'Actual location source'
  209 = 'Actual mirror position'
  220 = 'Actual motor current'
  211 = 'Actual motor offset'
  81 = 'Actual offset'
  78 = 'Actual position'
  224 = 'Actual positioning motor current'
  1079 = 'Actual positions'
  540 = 'Actual pressure setpoint'
  503 = 'Actual target'
  392 = 'Actual time source'
  1022 = 'Actual top setpoint:'
  1528 = 'Actual torque feedback'
  1879 = 'Actual velocity'
  421 = 'Actual:'
  1624 = 'actVelo'
  1942 = 'ActVelo'
  1839 = 'Add offset'
  125 = 'ADMIN'
  127 = 'Admin'
  1260 = 'Administrate'
  1543 = 'Advanced'
  1147 = 'Advanced status'
  963 = 'Afer the system is rebooted, you will see a Microsoft Windows environment.'
  567 = 'Alarm config:'
  518 = 'Alarm enabled'
  807 = 'All OK'
  1999 = 'Allow an observer to go to this position'
  1997 = 'Allow an observer to go to this position by using the GUI'
  1998 = 'Allow an observer to go to this position by using the GUI buttons'
  422 = 'Allowed'
  423 = 'Allowed:'
  1996 = 'allowObserver'
  1369 = 'Alpha'
  1608 = 'alpha'
  1925 = 'Alpha and delta'
  1861 = 'Alpha offset'
  1372 = 'Alpha proper motion'
  1871 = 'Alpha travelled so far'
  1859 = 'Alpha velocity'
  1089 = 'Alternatively, go to the termal position of another instrument:'
  1088 = 'Alternatively, go to the termal position of other instruments:'
  391 = 'Altitude'
  348 = 'Always use local clock istead of PTP'
  351 = 'Always use local clock istead of the PTP (IEEE1588) clock'
  349 = 'Always use position below istead of from GPS'
  350 = 'Always use position from config instead of from GPS'
  343 = 'Always use the local clock'
  345 = 'Always use the local clock (even \nif a more accurate one is available)'
  346 = 'Always use the local clock (even if\na more accurate one is available)'
  344 = 'Always use the local clock (even if a more accurate one is available)'
  347 = 'Always use the local clock istead of PTP'
  352 = 'Always use the local clock istead of the PTP (IEEE1588) clock'
  355 = 'Always use the location from the config instead of from the GPS'
  353 = 'Always use the position from config instead of from GPS'
  354 = 'Always use the position from the config instead of from the GPS'
  168 = 'AMS NetId'
  1453 = 'AN'
  793 = 'AND'
  1933 = 'and'
  832 = 'AND\n(7s timeout)'
  834 = 'AND\n7 sec\ntimeout'
  833 = 'AND\n7s timeout'
  835 = 'AND\nwith 7 sec\ntimeout'
  587 = 'and:  AxialForce = 390 daN * sin(elevation)'
  588 = 'and:  AxialForce = 390 daN * sin(Elevation)'
  586 = 'and:  AxialPressureSetpoint = CorrectionCoefficient * AxialForce / 18'
  584 = 'and: AxialPressureSetpoint = CorrectionCoefficient * AxialForce / 18'
  155 = 'ANTI-B DRIVE'
  246 = 'Anti-backlash'
  248 = 'Anti-backlash\n(ABL)'
  247 = 'Anti-backlash\nABL)'
  91 = 'Anti-backlash\naxis'
  99 = 'Anti-backlash\ndrive'
  1697 = 'Anti-backlash axis (ABL)'
  1070 = 'Anti-backlash lifted'
  252 = 'Anti-backlash motor\n(ABL)'
  1696 = 'Anti-backlash motor (ABL)'
  226 = 'Anti-backlash motor actual current'
  1025 = 'Apply'
  609 = 'Apply new value'
  1911 = 'Apply offsets'
  2040 = 'apply the following offset to the active rotator'
  2042 = 'apply the following offset to the Cassegrain rotator'
  2041 = 'apply the following offset to the Cassegrainrotator'
  2043 = 'apply the following offset to the Nasmyth rotator'
  1376 = 'arcsec'
  1870 = 'arcsec / h'
  1869 = 'arcsec / s'
  2055 = 'At fixed position:'
  739 = 'at high speed'
  738 = 'at low speed'
  736 = 'at low speed!'
  244 = 'At position'
  26 = 'Auto'
  1538 = 'AUTO'
  545 = 'AUTO pressure setpoint'
  554 = 'Automatic'
  552 = 'Automatic pressure setpoint'
  612 = 'Automatic pressure setpoint:'
  1456 = 'AUX1A'
  1478 = 'AUX1B'
  1118 = 'Average'
  1515 = 'Average 1 sec'
  232 = 'average current'
  2100 = 'Average error'
  1521 = 'Average error (1 sec)'
  1516 = 'Average error 1 sec'
  1520 = 'Average error last sec'
  604 = 'Average of force sensors alarms [daN]'
  603 = 'Average of force sensors alarms [daN]\n(SO)'
  631 = 'Average of force sensors [daN]'
  2098 = 'Avg error'
  1455 = 'AW'
  1145 = 'Awake'
  1444 = 'Awake axes'
  1513 = 'Axes'
  621 = 'Axial pressure\n@ mirror cell'
  622 = 'Axial pressure\n@ regulator'
  625 = 'Axial regulator'
  628 = 'Axial regulator\nfeedback'
  627 = 'Axial regulator\nmeasured'
  626 = 'Axial regulator\nsetpoint'
  654 = 'Axial support automatic control'
  647 = 'Axial support controller input'
  648 = 'Axial support controller inputs'
  644 = 'Axial support setpoint selection'
  156 = 'Axis'
  23 = 'Axis status'
  1751 = 'Az'
  1754 = 'az'
  1472 = 'Az centering error (cos component)'
  1470 = 'Az centering error (sin component)'
  1477 = 'Az change supplied through auxiliary reading 1'
  1612 = 'azi'
  1652 = 'AZI'
  1830 = 'AZI Average error (1 sec)'
  2005 = 'AZI position to go to, in degrees'
  1831 = 'AZI RMS error (1 sec)'
  1383 = 'Azimuth'
  1618 = 'azimuth'
  2110 = 'Azimuth %.0f°'
  1908 = 'Azimuth and elevation'
  1546 = 'Azimuth axis'
  813 = 'Azimuth axis release'
  1545 = 'Azimuth axus'
  2000 = 'Azimuth position to go to'
  2001 = 'Azimuth position to go to (absolute position, in degrees)'
  2002 = 'Azimuth position to go to, in degrees'
  816 = 'Azimuth release'
  815 = 'Azimuth release OK'
  1888 = 'Azimuth step'
  1891 = 'Azimuth step size'
  812 = 'AzimuthRelease'
  1613 = 'azi_start'
  1586 = 'B'
  284 = 'b:'
  1071 = 'Backlash lifted'
  994 = 'Bearing temperature [°C]'
  1506 = 'Bipolar torque limit'
  1509 = 'Bipolar torque limit (in %)'
  1736 = 'Bistable'
  1214 = 'Bit length (1 bit = x milliseconds)'
  1215 = 'Bit length (x where 1 bit = x milliseconds)'
  1212 = 'Bit pattern (bit high = alert active)'
  1264 = 'Blank screen'
  34 = 'BOTTOM'
  427 = 'Bottom'
  956 = 'BOTTOM\n5'
  957 = 'Bottom\n5'
  958 = 'Bottom\n6'
  959 = 'Bottom\n7'
  960 = 'Bottom\n8'
  782 = 'BOTTOM 1'
  788 = 'Bottom 1'
  789 = 'Bottom 5'
  938 = 'Bottom 5 no underpressure'
  847 = 'Bottom 5 underpressure'
  882 = 'Bottom 5 underpressure OK'
  790 = 'Bottom 6'
  939 = 'Bottom 6 no underpressure'
  848 = 'Bottom 6 underpressure'
  883 = 'Bottom 6 underpressure OK'
  791 = 'Bottom 7'
  940 = 'Bottom 7 no underpressure'
  849 = 'Bottom 7 underpressure'
  884 = 'Bottom 7 underpressure OK'
  792 = 'Bottom 8'
  941 = 'Bottom 8 no underpressure'
  850 = 'Bottom 8 underpressure'
  885 = 'Bottom 8 underpressure OK'
  1334 = 'Bottom and top pumps relay:'
  945 = 'Bottom no overpressure'
  943 = 'Bottom no overpressure OK'
  856 = 'Bottom overpressure'
  887 = 'Bottom overpressure OK'
  985 = 'Bottom setpoint:'
  891 = 'Bottom TRIP OK'
  747 = 'Brake'
  1293 = 'Brake release'
  1537 = 'Brake state'
  169 = 'Bus NetId'
  1737 = 'Buttons'
  1151 = 'Buzzer is sounding'
  962 = 'By pressing the REBOOT button below, you will reboot the whole Mercator\nTelescope Control System. This takes approximately 3 minutes.'
  1178 = 'Bypass briefly'
  1180 = 'Bypass for %.0f seconds'
  1179 = 'Bypass for %.1f seconds'
  1181 = 'Bypass permanently\n\n(until re-initialization)'
  1176 = 'Bypass permanently\n(until re-initialization)'
  1161 = 'Bypass permanently\n(until Safety is re-initialized)'
  1162 = 'Bypass sensors permanently\n(until Safety is re-initialized)'
  1208 = 'Bypassing time after entering password'
  1209 = 'Bypassing time after entering password (s)'
  1210 = 'Bypassing time after entering password (sec)'
  1211 = 'Bypassing time after entering password [s]'
  106 = 'byte(s)'
  657 = 'c'
  658 = 'C'
  1761 = 'C++ task status'
  1451 = 'CA'
  237 = 'Calibrate'
  238 = 'Calibration'
  489 = 'Calibration move to 0 torque vel. [°/s]'
  485 = 'Calibration move to 0 torque velocity [°/s]'
  488 = 'Calibration offset [°]'
  487 = 'Calibration range [°]'
  484 = 'Calibration start position [°]'
  486 = 'Calibration velocity [°/s]'
  289 = 'CAN state'
  287 = 'CAN state (dec, hex, bin):'
  288 = 'CAN state (decimal, hex, bin):'
  278 = 'CAN state:'
  324 = 'Cancel'
  274 = 'CANopen'
  275 = 'CANopen bus'
  115 = 'CANopen bus NetID'
  114 = 'CANopen NetID'
  116 = 'CANopen node port'
  304 = 'CAS'
  307 = 'Cas'
  1912 = 'cas'
  161 = 'Cassegrain'
  504 = 'CASSEGRAIN'
  1940 = 'Cassegrain\nrotation'
  1906 = 'Cassegrain rotation'
  1962 = 'Cassegrain rotation (%s)'
  1957 = 'Cassegrain rotator'
  1958 = 'Cassegrain rotator (%s)'
  1961 = 'Cassegrain rotator name (e.g. name of the instrument)'
  1902 = 'Cassegrain step'
  1897 = 'Cassegrain step size'
  746 = 'CCW'
  1040 = 'CCW direction'
  1041 = 'CCW sense of direction'
  710 = 'centre'
  663 = 'Change ...'
  1021 = 'Change frequencies manually'
  1428 = 'Change instrument ...'
  1277 = 'Change M3'
  1422 = 'Change operator ...'
  660 = 'Change operator to:'
  608 = 'Change setpoint'
  1317 = 'Change the instrument'
  1326 = 'Change the instrument instrument'
  1429 = 'Change the instrument to:'
  1498 = 'Channel peak current'
  1499 = 'Channel rated current'
  1434 = 'Checkbox'
  409 = 'Checksum status'
  975 = 'Chiller'
  1168 = 'Circuit 1'
  1030 = 'Circulation pump relay:'
  1953 = 'click'
  766 = 'Clockwis'
  764 = 'Clockwise'
  1303 = 'Clockwise (CW)'
  65 = 'Close'
  1330 = 'Close window'
  47 = 'closed'
  59 = 'Closed position [°]'
  46 = 'Closed position:'
  39 = 'Closing velocity [°/s]'
  471 = 'Closing velocity:'
  1005 = 'Coefficient a'
  1006 = 'Coefficient b'
  1007 = 'Coefficient c'
  901 = 'COM'
  898 = 'COM error'
  826 = 'COM/FB/OUT'
  1094 = 'Command'
  1032 = 'Command the safety'
  2073 = 'Commands'
  823 = 'Communication'
  899 = 'Communication error'
  36 = 'CONFIG'
  1258 = 'Configure ...'
  1261 = 'Configure MTCS ...'
  359 = 'Configured location: altitude [meters above sea level]'
  358 = 'Configured location: latitude [°, positive = E, negative = W]'
  356 = 'Configured location: longitude [degrees]'
  357 = 'Configured location: longitude [°, positive = N, negative = S]'
  1223 = 'Confirm'
  1635 = 'Constant vertical displacement'
  117 = 'Continuous current limit'
  177 = 'Control'
  989 = 'Control loop cycle time [s]'
  988 = 'Control loop cycle tine'
  990 = 'Control loop hysteresis [Hz]'
  656 = 'Controller feedback:'
  593 = 'Controller integral time (Tn) [s]'
  591 = 'Controller Kp [bar/daN]'
  594 = 'Controller maximum output limit [bar]'
  595 = 'Controller minimum output limit [bar]'
  592 = 'Controller proportional factor (Kp) [bar/daN]'
  655 = 'Controller setpoint:'
  577 = 'Correction coefficient'
  582 = 'Correction coefficient [unitless]'
  1575 = 'Counter overflow'
  1569 = 'Counter underflow'
  1568 = 'Counter value:'
  767 = 'Counter-clockwise'
  1042 = 'Counter-clockwise (CCW)'
  192 = 'Couple'
  188 = 'Coupling'
  68 = 'COVER'
  71 = 'Cover'
  520 = 'Critically high'
  519 = 'Critically low'
  1936 = 'Cumulative offset'
  1938 = 'Cumulative offsets'
  457 = 'Current'
  451 = 'Current (0-8 panels!):'
  450 = 'Current (all 8 panels!):'
  449 = 'Current measurement (all 8 panels!)'
  379 = 'Current time source'
  676 = 'Currents'
  765 = 'CW'
  70 = 'd'
  2083 = 'D'
  1611 = 'd(alpha)/dt'
  1875 = 'd/m/s'
  286 = 'd:'
  1246 = 'DA: Dome Access cabinet'
  1049 = 'Data'
  367 = 'Date & time'
  366 = 'Date / time'
  378 = 'Date and time'
  1745 = 'Dec.'
  290 = 'dec:'
  1397 = 'Declination'
  193 = 'Decouple'
  1310 = 'Default positions'
  1370 = 'Delta'
  1609 = 'delta'
  1862 = 'Delta offset'
  1373 = 'Delta proper motion'
  1872 = 'Delta travelled so far'
  1343 = 'Delta UT (UT1 - UTC)'
  1860 = 'Delta velocity'
  2038 = 'Derotator\noffsets'
  2082 = 'Derotator active'
  2057 = 'Derotator active:'
  2036 = 'Derotators'
  533 = 'Dewpoints'
  1973 = 'Diagnostic number'
  1974 = 'Diagnostic number S-0-390'
  50 = 'diff %.2f°'
  443 = 'Diff: %.2f°'
  88 = 'Difference'
  329 = 'Difference '
  218 = 'Difference (<0.001° = OK)'
  216 = 'Difference (<1'
  217 = 'Difference (<1° = OK)'
  1530 = 'Digital inputs'
  1531 = 'Digital inputs / output'
  1532 = 'Digital inputs / outputs'
  1533 = 'Digital outputs'
  1481 = 'Disable'
  1157 = 'Disable alarm permanently\n(until Safety is re-initialized)'
  1591 = 'Disable C reset'
  1206 = 'Disable Dome Access control permanently'
  1204 = 'Disable Dome Access permanently'
  1158 = 'Disable door sensors permanently\n(until Safety is re-initialized)'
  1160 = 'Disable permanently\n(until Safety is re-initialized)'
  14 = 'Disabled'
  914 = 'Discrepancy\nerror'
  913 = 'DiscrepancyError'
  670 = 'Dismiss'
  1329 = 'Dismiss window'
  418 = 'Distance between panels:'
  1880 = 'Distance travelled so far'
  1446 = 'Do homing'
  1276 = 'Do initial thermal focus'
  136 = 'Do rotatiob'
  137 = 'Do rotation'
  140 = 'Do translation'
  1430 = 'Do you want to (re)initialize the whole Telescope Control System?'
  1425 = 'Do you want to make the telescope go to sleep?'
  1424 = 'Do you want to wake up the telescope?'
  802 = 'Dome'
  1119 = 'Dome Access'
  1194 = 'Dome access'
  1203 = 'Dome access control is disabled permanently'
  1201 = 'Dome access summary'
  1159 = 'Dome sensors'
  475 = "Don't show the timing status as ERROR in case the serial link fails"
  1148 = 'Door 1 is closed'
  1149 = 'Door 2 is closed'
  1191 = 'Door sensors'
  1195 = 'Doors not opened'
  1240 = 'Doors were opened'
  1190 = 'Doors were opened without bypass'
  1189 = 'Doors were opened without password'
  322 = 'Draw mirror as cassegrain below [mm]'
  323 = 'Draw mirror as nasmyth above [mm]'
  321 = 'Draw mirror as nasmyth below [mm]'
  320 = 'Draw mirror as nasmyth below: [mm]'
  319 = 'Draw mirror in nasmyth position limit  [mm]'
  433 = 'Drawing angle'
  435 = 'Drawing angle (offset) [°]'
  434 = 'Drawing angle [°]'
  157 = 'Drive'
  749 = 'Drive Brake'
  750 = 'Drive brake'
  748 = 'Drive CCW'
  1301 = 'Drive CW'
  745 = 'Drive enable'
  1978 = 'Drive in safe (= blocked) state'
  1975 = 'Drive in safe state'
  1976 = 'Drive in safe state (orange = blocked)'
  1977 = 'Drive in safe state (safe = blocked)'
  1283 = 'Drive release'
  1494 = 'Drives'
  1769 = 'ds'
  2084 = 'E'
  1548 = 'E 90'
  1549 = 'E 90°'
  1349 = 'Earth polar motion X in degrees'
  1351 = 'Earth polar motion X [degrees]'
  1350 = 'Earth polar motion Y in degrees'
  1352 = 'Earth polar motion Y [degrees]'
  1475 = 'ECEC'
  1473 = 'ECES'
  551 = 'Edit'
  547 = 'Edit ...'
  42 = 'Editable'
  3 = 'Editable\nconfig'
  1752 = 'El'
  1476 = 'El centering error (cos component)'
  1474 = 'El centering error (sin component)'
  1616 = 'ele'
  1651 = 'ELE'
  1832 = 'ELE Average error (1 sec)'
  2007 = 'ELE position to go to, in degrees'
  1833 = 'ELE RMS error (1 sec)'
  1384 = 'Elevation'
  1619 = 'elevation'
  2111 = 'Elevation %.0f(°'
  2112 = 'Elevation %.0f°'
  1792 = 'Elevation axis'
  1237 = 'Elevation axis release'
  1889 = 'Elevation step'
  1890 = 'Elevation step size'
  919 = 'Emergency \nstop\n@ dome'
  918 = 'Emergency \nstop @ dome'
  922 = 'Emergency stop\n@ control room'
  920 = 'Emergency stop\n@ dome'
  1234 = 'Emergency stop\n@ dome (1)'
  1236 = 'Emergency stop\n@ dome (no. 1)'
  1235 = 'Emergency stop\n@ dome (no. 2)'
  1233 = 'Emergency stop\n@ dome 1'
  1200 = 'Emergency stop\n@ dome access'
  921 = 'Emergency stop\n@ first floor'
  917 = 'Emergency stop@ dome'
  799 = 'Emergency stops'
  808 = 'Emergency stops OK'
  929 = 'Emergency stops summary'
  446 = 'Enable'
  1483 = "Enable '%s' "
  560 = 'Enable automatic'
  1590 = 'Enable C reset'
  1589 = 'Enable counter reset C'
  561 = 'Enable fixed'
  678 = 'Enable keypad'
  1480 = 'Enable or disable this model'
  1479 = 'Enable/disable'
  13 = 'Enabled'
  441 = 'enabled'
  672 = 'Encoder error signal:'
  741 = 'Encoder offset (encoder ticks for z = 0mm)'
  740 = 'Encoder offset (no. of encoder ticks for z = 0mm)'
  1053 = 'Encoder value'
  205 = 'Encoder-to-mirror ratio'
  1544 = 'Encoders'
  2088 = 'End of travel reache'
  2089 = 'End of travel reached'
  667 = 'Enter password if needed:'
  1404 = 'Epoch'
  1379 = 'Epoch and equinox'
  801 = 'Error'
  2097 = 'Error (1 sec)'
  1529 = 'Error C1D'
  24 = 'Error ID'
  162 = 'Error id:'
  113 = 'EtherCAT NetID'
  1457 = 'EW misalignment of azimuth axis'
  337 = 'EXT: %s'
  1583 = 'Extern latch status'
  841 = 'External'
  842 = 'External\nDevice\nMonitor'
  362 = 'External timestamp'
  365 = 'EXTERNAL: %s'
  1578 = 'Extrapolation stall'
  731 = 'FALSE if the motor final sense must be CounterClockWise (+ motion on the screw), TRUE if the motor final sense must be ClockWise (- motion on the screw) (for Z axis: at low speed)'
  1728 = 'FAST'
  1297 = 'Fast (<<< or >>>) if backlash must not be lifted'
  1296 = 'Fast (>>>) if backlash must not be lifted'
  1299 = 'Faster (<<< or >>>) in the direction of no backlash'
  1300 = 'Faster (<<< or >>>) in the direction without backlash'
  1294 = 'Fault signak'
  751 = 'Fault signal'
  902 = 'FB'
  1784 = 'Feedback'
  818 = 'Filter'
  1717 = 'Filter wheel'
  727 = 'Final sense (False = CCW, True = CW)'
  1064 = 'Final sense (True = CCW, False = CW)'
  1302 = 'Final sense (True = CW, False = CCW)'
  803 = 'First floor'
  2054 = 'Fixed position:'
  1308 = 'Fixed positions'
  553 = 'Fixed pressure setpoint'
  611 = 'Fixed pressure setpoint:'
  1634 = 'FLOP'
  1806 = 'for'
  1058 = 'Force'
  1812 = 'FORCE\nLOCK'
  1813 = 'FORCE\nUNLOCK'
  650 = 'Force feedback:'
  1055 = 'Force move'
  649 = 'Force setpoint:'
  1050 = 'Frame'
  1051 = 'Frames'
  843 = 'Frequency\nrises'
  844 = 'Frequency\nrises during \nstartup\n(QMin -> 0)'
  858 = 'Frequency \nrises\nduring \nstartup\n\n(QMin -> 0)'
  857 = 'Frequency \nrises during \nstartup\n(QMin -> 0)'
  1001 = 'Frequency measurement full scale [Hz]'
  1004 = 'Frequency measurement [Hz]'
  859 = 'Frequency rises\nduring startup\n(QMin -> 0)'
  924 = 'Frequency rising'
  864 = 'Frequency rising\nerror'
  862 = 'Frequency rising\nerror\n(QMin -> 0)'
  866 = 'Frequency rising \nerror'
  923 = 'Frequency rising after startup'
  926 = 'Frequency rising at startup'
  867 = 'Frequency rising error'
  1009 = 'Frequency[Hz] = a * BearingTemperature[Celsius]^2 + b * BearingTemperature[Celsius] + c'
  1008 = 'Frequency[Hz] = a * temp[Celsius]^2 + b * temp[Celsius] + c'
  971 = 'Full reset\n(REBOOT)'
  1265 = 'Full reset\n(REBOOT) ...'
  1263 = 'Full reset ...\n(REBOOT)'
  900 = 'Function block'
  904 = 'Function Blocks'
  1587 = 'Gate'
  190 = 'Gear IN'
  191 = 'Gear Out'
  189 = 'Gearing'
  132 = 'GENERAL'
  152 = 'General'
  37 = 'General settings'
  1187 = 'General statis'
  1188 = 'General status'
  403 = 'Geoid  separation'
  17 = 'GO'
  664 = 'Go'
  198 = 'Go to'
  159 = 'Go to %S'
  160 = 'Go to %s'
  511 = 'Go to ...'
  1325 = 'Go to instrument'
  200 = 'Go to new position'
  199 = 'Go to position'
  1410 = 'Go to sleep'
  1426 = 'Go to sleep ...'
  1085 = 'Go to this position'
  1086 = 'Go to this thermal position'
  483 = 'Goto offset velocity [°/s]'
  481 = 'Goto offset velocity [°]'
  478 = 'Goto position improving time [s]'
  479 = 'Goto position velocity'
  480 = 'Goto position velocity [mm/s]'
  513 = 'Goto procedure'
  482 = 'Goto target velocity [°/s]'
  1345 = 'GPS data'
  394 = 'GPS info'
  405 = 'GPS status'
  1773 = 'h'
  1873 = 'h/m/s'
  1876 = 'h/m/s *'
  1874 = 'h/m/s and d/m/s'
  285 = 'h:'
  1658 = 'Hardware limit switches'
  2109 = 'Health'
  564 = 'Health status'
  1039 = 'Heat exchanger'
  1099 = 'Heater'
  1346 = 'Height above sea level'
  67 = 'HERMES'
  521 = 'High'
  1964 = 'High enough'
  1315 = 'High frequency (QMin)'
  1256 = 'High speed'
  769 = 'High speed (Z axis only!)'
  762 = 'High speed (Z only!)'
  763 = 'High speed (Z only)'
  590 = 'Hint:  AxialPressure = CorrectionCoefficient * AxialForce / 18'
  585 = 'Hint:  AxialPressureSetpoint = CorrectionCoefficient * AxialForce / 18'
  583 = 'Hint: AxialPressureSetpoint = CorrectionCoefficient * AxialForce / 18'
  581 = 'Hint: RadialPressureSetpoint = CorrectionCoefficient * 1.33 bar * cos(elevation)'
  589 = 'Hint: RadialPressureSetpoint = CorrectionCoefficient * 1.33 bar * cos(Elevation)'
  580 = 'Hint: with: RadialPressureSetpoint = CorrectionCoefficient * 1.33 bar * cos(elevation)'
  2079 = 'HMI (GUI) instrument angle for drawing ROC'
  2080 = 'HMI (GUI) instrument angle for drawing RON'
  2078 = 'HMI (GUI) instrument angle for ROC'
  1952 = 'hold'
  69 = 'HOME'
  673 = 'Home'
  184 = 'Home Switch'
  272 = 'Homing'
  254 = 'Homing Cont. current limit'
  256 = 'Homing cont. current limit'
  257 = 'Homing cont. current limit (mA)'
  260 = 'Homing cont. current limit [mA]'
  255 = 'Homing peak current limit'
  258 = 'Homing peak current limit [mA['
  259 = 'Homing peak current limit [mA]'
  268 = 'Homing search limit switch  velocity [mm/s]'
  490 = 'Homing search limit switch vel. [mm/s]'
  185 = 'Homing Switch'
  491 = 'Homing to hardware stop vel. [mm/s]'
  269 = 'Homing to hardware stop velocity [mm/s]'
  267 = 'Homing velocity [mm/s]'
  271 = 'Hominh'
  402 = 'Horizontal dilution of position'
  1461 = 'Horizontal displacement of Nasmyth rotator'
  1400 = 'Hour Angle'
  1655 = 'How many degrees should the moveOutOfLimitSwitch process try to move?'
  1245 = 'HS: Hydraulics & Safety panel'
  775 = 'Hydraulics'
  949 = 'Hydraulics error'
  876 = 'Hydraulics health'
  814 = 'Hydraulics OK'
  1015 = 'Hydraulics safety'
  1020 = 'Hydraulics safety (see Safety tab for details!)'
  1019 = 'Hydraulics safety (see Safety tab for more!)'
  875 = 'Hydraulics summary'
  35 = 'I/O'
  1449 = 'IA'
  1447 = 'IE'
  476 = 'Ignore  serial link errors for overall Timing status'
  1567 = 'Incremental encoder'
  101 = 'Index'
  1450 = 'Index error in azimuth'
  1448 = 'Index error in elevation'
  8 = 'InfoData:'
  685 = 'Initialization'
  10 = 'Initialize'
  1603 = 'Input'
  1579 = 'Input A status'
  1580 = 'Input B status'
  1581 = 'Input C status'
  1582 = 'Input gate status'
  1576 = 'Input status'
  1093 = 'Instrument'
  1413 = 'INSTRUMENT'
  1266 = 'Instrument 0'
  1267 = 'Instrument 1'
  1268 = 'Instrument 2'
  1269 = 'Instrument 3'
  1270 = 'Instrument 4'
  1271 = 'Instrument 5'
  1272 = 'Instrument 6'
  1273 = 'Instrument 7'
  1274 = 'Instrument 8'
  1275 = 'Instrument 9'
  336 = 'INT: %s'
  361 = 'Internal timestamp'
  364 = 'INTERNAL: %s'
  1780 = 'INVALID'
  75 = 'IO'
  1083 = 'is '
  1082 = 'is:'
  1913 = 'Joystick\nAZI & ELE'
  1916 = 'Joystick\nAZI / ELE'
  1914 = 'Joystick\nROC & RON'
  1917 = 'Joystick\nROC / RON'
  1836 = 'Joystick AZI & ELE'
  1837 = 'Joystick ROC & RON'
  1389 = 'Julian Date (JD)'
  1390 = 'Julian Day (JD)'
  1378 = 'km/s'
  133 = 'KNOWN'
  134 = 'KNOWN\nPOSITIONS'
  1834 = 'Known positions'
  1318 = 'Label'
  1169 = 'Lamps circuit 1'
  1170 = 'Lamps circuit 2'
  1171 = 'Lamps circuit 3'
  1172 = 'Lamps circuit 4'
  1192 = 'Lamps circuits'
  1153 = 'Lamps relay 1 is closed'
  1154 = 'Lamps relay 2 is closed'
  1155 = 'Lamps relay 3 is closed'
  1156 = 'Lamps relay 4 is closed'
  1193 = 'Lamps relays'
  1167 = 'Lamps status'
  1385 = 'LAST'
  1097 = 'Last known positions'
  1588 = 'Latch'
  1570 = 'Latch C Valid'
  1572 = 'Latch C valid'
  1571 = 'Latch extern Valid'
  1573 = 'Latch extern valid'
  390 = 'Latitude'
  1344 = 'Leap seconds (TAI - UTC)'
  1592 = 'LIDA 1'
  1593 = 'LIDA 2'
  1594 = 'LIDA 3'
  1595 = 'LIDA 4'
  1597 = 'LIDA summary'
  187 = 'Limit switch polarity'
  186 = 'Limit switch positive edge'
  178 = 'Limit switches'
  1667 = 'Limit the maximum acceleration/deceleration of the physical axis to this value in degrees/sec'
  1668 = 'Limit the maximum acceleration/deceleration of the physical axis, in degrees/sec^2'
  1665 = 'Limit the maximum position of the physical axis to this value in degrees'
  1663 = 'Limit the maximum position of the virtual axis to this value in degrees'
  1666 = 'Limit the maximum velocity of the physical axis to this value in degrees/sec'
  1661 = 'Limit the minimum position of the axis to this value in degrees, of the virtual axis'
  1664 = 'Limit the minimum position of the physical axis to this value in degrees'
  1662 = 'Limit the minimum position of the virtual axis to this value in degrees'
  2044 = 'Limits during tracking and pointing'
  0 = 'LOAD'
  2028 = 'Load the pointing model with the same name as above'
  1360 = 'Local pressure, fixed by config [hectoPascal = millibar]'
  1357 = 'Local temperatu'
  1359 = 'Local temperature, fixed by config [degrees]'
  388 = 'Location'
  1540 = 'LOCK'
  49 = 'locked'
  659 = 'Log in as:'
  682 = 'Log out'
  665 = 'Login'
  669 = 'LOGIN FAILED'
  389 = 'Longitude'
  522 = 'Low'
  846 = 'Low frequency \n(QMin)'
  845 = 'Low frequency (QMin)'
  725 = 'm'
  954 = 'M'
  253 = 'M3'
  221 = 'mA'
  437 = 'magnet'
  465 = 'Magnets'
  447 = 'Magnets relay'
  453 = 'Magnets relay (4 panels):'
  452 = 'Magnets relay (all 4 panels):'
  448 = 'Magnets relay:'
  40 = 'Magnets remanent time [s]'
  66 = 'MAIA'
  27 = 'Manual'
  2074 = 'Manual commands'
  546 = 'MANUAL pressure setpoint'
  1065 = 'Margin when moving before the final move'
  300 = 'Max offset error [°]'
  303 = 'Max position error [mm]'
  299 = 'Max position error [°]'
  181 = 'Max profile velocity'
  19 = 'Max velocity'
  1674 = 'Maximum acceleration of the physical axis, in degrees/sec^2'
  1676 = 'Maximum acceleration of the physical axis, in degrees/sec^2 (always >0)'
  1677 = 'Maximum acceleration or deceleration of the physical axis, in degrees/sec^2 (>0)'
  1721 = 'Maximum distance to be covered while searching for the homing mark, in degrees'
  997 = 'Maximum output frequency [Hz]'
  605 = 'Maximum output limit [bar]'
  2047 = 'Maximum pointing and tracking setpoint of the axis in degrees (a bit before the soft limit)'
  2046 = 'Maximum position and tracking setpoint of the axis in degrees (a bit before the soft limit)'
  1672 = 'Maximum position limit of the physical axis in degrees'
  1670 = 'Maximum position limit of the virtual axis to this value in degrees'
  1673 = 'Maximum velocity limit of the physical axis in degrees/sec'
  1678 = 'Maximum velocity limit of the physical axis in degrees/sec (>0)'
  1675 = 'Maximum velocity limit of the physical axis in degrees/sec (always >0)'
  996 = 'Maximumoutput frequency [Hz]'
  297 = 'maxPositionError ['
  298 = 'maxPositionError [°]'
  987 = 'measured:'
  630 = 'Measurement\nenabled'
  1031 = 'Measurement\noffset'
  1028 = 'Measurements'
  1729 = 'MEDIUM'
  531 = 'Mercator'
  675 = 'Mercator\nTelescope \nControl System'
  532 = 'Mercator\nTelescope Control System'
  1653 = 'MEROPE'
  1102 = 'mG'
  243 = 'Min. current'
  415 = 'Min. distance between panels [°]'
  1316 = 'Min. frequency (QMin)'
  242 = 'Minimum current'
  425 = 'Minimum distance between panels:'
  995 = 'Minimum output frequency [Hz]'
  606 = 'Minimum output limit [bar]'
  2045 = 'Minimum pointing and tracking setpoint of the axis in degrees (a bit before the soft limit)'
  1671 = 'Minimum position limit of the physical axis in degrees'
  1669 = 'Minimum position limit of the virtual axis to this value in degrees'
  998 = 'Minimum pressure [Hz]'
  728 = 'Minimum steps for final move'
  424 = 'Minimum:'
  711 = 'mirrorCell'
  717 = 'mirrorCell * mirrorCellTemperature'
  328 = 'mm'
  1484 = 'Model 0'
  1485 = 'Model 1'
  1486 = 'Model 2'
  1487 = 'Model 3'
  1488 = 'Model 4'
  1489 = 'Model 5'
  1490 = 'Model 6'
  1491 = 'Model 7'
  1492 = 'Model 8'
  1493 = 'Model 9'
  179 = 'Modes of operation'
  1386 = 'Modified Julian Date (MJD)'
  1391 = 'Modified Julian Day (MJD)'
  868 = 'Monitor'
  896 = 'Monitor    '
  1735 = 'Monostable'
  395 = 'More GPS info'
  2076 = 'Motion'
  1252 = 'Motion allowed'
  931 = 'Motion blocking'
  930 = 'Motion blocking summary'
  1197 = 'Motion not blocked'
  1196 = 'Motion release'
  327 = 'Motor average current'
  1502 = 'Motor continous stall current'
  1500 = 'Motor continous stall torque'
  466 = 'Motor current'
  468 = 'Motor relay:'
  204 = 'Motor-to-mirror ratio'
  1443 = 'Move'
  20 = 'Move absolute'
  1622 = 'move absolute'
  2048 = 'Move absolute (virtual)'
  1841 = 'move active rotator'
  1846 = 'move active rotator(s)'
  1319 = 'Move after initialization'
  1312 = 'Move axes'
  2004 = 'Move AZI (TRUE) or not (FALSE)'
  1840 = 'move azimuth'
  2003 = 'Move azimuth (TRUE) or not (FALSE)'
  1844 = 'move azimuth axis'
  1945 = 'Move back to 0'
  1843 = 'move Cassegrain rotator'
  1073 = 'Move command'
  2006 = 'Move ELE (TRUE) or not (FALSE)'
  1845 = 'move elevation axis'
  1842 = 'move Nasmyth rotator'
  1646 = 'Move out <--'
  1643 = 'Move out <<<'
  1647 = 'Move out >>>'
  1814 = 'Move out of limit switch'
  1074 = 'Move procedure'
  1626 = 'move relativ'
  1063 = 'Move relative'
  1627 = 'move relative'
  2008 = 'Move ROC (TRUE) or not (FALSE)'
  2010 = 'Move RON (TRUE) or not (FALSE)'
  760 = 'Move steps'
  1075 = 'Move steps procedure'
  2037 = 'move the active derotator'
  2039 = 'move the active derotator with this offset'
  2035 = 'move the active rotator'
  1946 = 'Move to\nAZI / ELE / ROT'
  1947 = 'Move to fixed\nAZI / ELE / ROT'
  2018 = 'Move to the known position below'
  2019 = 'Move to the known position below before turning off derotators'
  2020 = 'Move to this known position (see choice above)'
  1320 = 'Move to this position after initialization'
  240 = 'Move velocity'
  2050 = 'Move Virtual  relative'
  2049 = 'Move Virtual absolute'
  2051 = 'Move Virtual relative'
  2052 = 'Move Virtual velocity'
  1096 = 'Move Z'
  1098 = 'Move Z axis'
  1251 = 'Movement allowed'
  1143 = 'MOVING'
  1144 = 'Moving'
  1259 = 'MTCS'
  1262 = 'MTCS config ...'
  1762 = 'Mu alpha'
  1763 = 'Mu Delta'
  1764 = 'Mu delta'
  752 = 'Multiplexer'
  1547 = 'N'
  1550 = 'N 0°'
  135 = 'Name'
  1468 = 'Name of the model (matched against the instrument name)'
  430 = 'Name of the panel set'
  1995 = 'Name of the position'
  305 = 'NasA'
  306 = 'NasB'
  316 = 'Nasmyth'
  317 = 'Nasmyth\nA'
  318 = 'Nasmyth\nB'
  492 = 'Nasmyth\nC'
  493 = 'Nasmyth\nD'
  1941 = 'Nasmyth\nrotation'
  494 = 'Nasmyth A'
  495 = 'Nasmyth B'
  496 = 'Nasmyth C'
  497 = 'Nasmyth D'
  1907 = 'Nasmyth rotation'
  1963 = 'Nasmyth rotation (%s)'
  1959 = 'Nasmyth rotator (%s)'
  1960 = 'Nasmyth rotator name (e.g. name of the instrument)'
  1901 = 'Nasmyth step'
  1896 = 'Nasmyth step size'
  538 = 'NE\n '
  1642 = 'Negative'
  182 = 'Negative Limit Switch'
  264 = 'Negative limit [mm]'
  214 = 'Negative soft limit'
  261 = 'Negative soft limit (mm)'
  262 = 'Negative soft limit [mm]'
  302 = 'Negative soft limit [°]'
  1512 = 'Negative torque limit'
  112 = 'NetID'
  111 = 'NetID\\'
  1026 = 'New bottom setpoint:'
  1024 = 'New setpoint:'
  1027 = 'New top setpoint:'
  610 = 'New value:'
  1282 = 'No fault'
  946 = 'No frequency rising error'
  944 = 'No overpressure'
  947 = 'No pressure rising error'
  1923 = 'No target'
  1922 = 'No target given'
  934 = 'No underpressure'
  948 = 'No underpressure error'
  1017 = 'No verpressure'
  276 = 'No. of boxes with error:'
  277 = 'No. of error boxes:'
  338 = 'No. of leap seconds'
  341 = 'No. of leap seconds (=UTC-TAI)'
  339 = 'No. of leap seconds (TAI to UTC)'
  340 = 'No. of leap seconds (UTC-TAI)'
  726 = 'No. of steps between braking and stopped'
  671 = 'No. of wrong passwords entered:'
  171 = 'Node Port'
  213 = 'None'
  1459 = 'Nonperpendicularity of azimuth and elevation axes'
  1452 = 'Nonperpendicularity of elevation and pointing axes'
  600 = 'North East sensor alarms [daN]\n(NE)'
  599 = 'North East sensor alarms [daN]\n(SO)'
  633 = 'North East sensor [daN]\n(NE)'
  602 = 'North West sensor alarms [daN]\n(NW)'
  601 = 'North West sensor alarms [daN]\n(SO)'
  634 = 'North West sensor [daN]\n(NW)'
  952 = 'NOT'
  870 = 'Not restarting'
  893 = 'Not stopping'
  194 = 'Not supported by this axis'
  195 = 'Not supported by this axis!'
  1877 = 'Note: 1 arcsecond = 15 seconds'
  1226 = 'Note: confirm button in\n GUI is \nonly enabled for staff'
  1227 = 'Note: confirm button in\n GUI is only enabled for staff'
  1225 = 'Note: confirm button in GUI\nis \nonly enabled for staff'
  1229 = 'Note: confirm button in GUI\nis only available to staff'
  1228 = 'Note: confirm button in GUI\nis only enabled for staff'
  1224 = 'Note: confirm button in GUI is \nonly enabled for staff'
  1221 = 'Note: GUI button is \nonly available to staff'
  1222 = 'Note: GUI button is \nonly enabled for staff'
  1129 = 'Note: only staff\ncan unblock from GUI'
  1130 = 'Note: only staff can\nunblock from GUI'
  1164 = 'Note: unblock from\nGUI is only available to staff)'
  1166 = 'Note: unblock from GUI\nis only available to staff'
  1165 = 'Note: unblock from GUI\nis only available to staff)'
  1163 = 'Note: unblock from GUI is'
  1458 = 'NPAE'
  1460 = 'NRX'
  1462 = 'NRY'
  1454 = 'NS misalignment of azimuth axis'
  396 = 'Number of satellites used'
  431 = 'Number of the panel set'
  1353 = 'Nutation adjustment dX [degrees]'
  1354 = 'Nutation adjustment dY [degrees]'
  536 = 'NW'
  537 = 'NW\n '
  1342 = 'Observatory location: altitude [meters above sea level]'
  1341 = 'Observatory location: latitude [°, positive = E, negative = W]'
  1407 = 'Observatory location: latitude [°, positive = N, negative = S]'
  1406 = 'Observatory location: longitude [°, positive = E, negative = W]'
  1340 = 'Observatory location: longitude [°, positive = N, negative = S]'
  1405 = 'Observatory location: longitude [°, ]'
  30 = 'Observer'
  661 = 'OBSERVER'
  1366 = 'Observing wavelength, fixed by config [microns]'
  197 = 'Offset'
  705 = 'offset'
  83 = 'Offset error'
  1898 = 'Offset in alpha / delta'
  1899 = 'Offset in azi / ele'
  1654 = 'Offset in degrees, of the absolute encoder, w.r.t. zero'
  1853 = 'Offset in degrees, of the motor encoder, w.r.t. zero'
  1835 = 'Offsets'
  1918 = 'Offsets\nAlpha / Delta / ROT'
  1920 = 'Offsets\nalpha / delta / ROT'
  1915 = 'Offsets\nAZI / ELE / ROT'
  1980 = 'offsetted'
  1900 = 'Offsetts in azi / ele'
  1910 = 'Offsetts in azi / ele / rot'
  1909 = 'Offsetts in azi / ele /rot'
  977 = 'Oil\nlevel'
  976 = 'Oil level'
  666 = 'OK'
  2086 = 'One ore more axes'
  2087 = 'One ore more axes\nreached their end of travel'
  48 = 'open'
  64 = 'Open'
  1577 = 'Open circuit'
  58 = 'Open position [°]'
  45 = 'Open position:'
  412 = 'OPENING'
  445 = 'Opening / closing'
  38 = 'Opening velocity [°/s]'
  470 = 'Opening velocity:'
  334 = 'Operator'
  874 = 'OR'
  1087 = 'Or, go to the termal position of other instruments:'
  1810 = 'Or, set the brake permanently:'
  308 = 'Other'
  309 = 'Other\n0'
  310 = 'Other\n1'
  311 = 'Other\n2'
  312 = 'Other\n3'
  313 = 'Other\n4'
  314 = 'Other\n5'
  315 = 'Other\n6'
  498 = 'Other 0'
  499 = 'Other 1'
  500 = 'Other 2'
  501 = 'Other 3'
  502 = 'Other 4'
  1183 = 'Other status'
  1182 = 'Otherstatus'
  903 = 'OUT'
  523 = 'Output 1'
  524 = 'Output 2'
  525 = 'Output 3'
  526 = 'Output 4'
  527 = 'Output 5'
  528 = 'Output 6'
  529 = 'Output 7'
  530 = 'Output 8'
  742 = 'Output A'
  743 = 'Output B'
  744 = 'Output C'
  543 = 'Output:'
  825 = 'Outputs'
  819 = 'Over\npressure'
  827 = 'Overpressure'
  1018 = 'Overpressure error'
  888 = 'Overpressure OK'
  32 = 'OVERVIEW'
  677 = 'Overview'
  1748 = 'P.a.'
  1756 = 'PA'
  1757 = 'pa'
  51 = 'Panel 1'
  52 = 'Panel 2'
  53 = 'Panel 3'
  54 = 'Panel 4'
  428 = 'Panel 5'
  432 = 'Panel settings'
  456 = 'Panel shown below'
  463 = 'Panels'
  455 = 'Panelset'
  458 = 'Panelset magnets'
  429 = 'Panelset settings'
  55 = 'Panelset settings for'
  1375 = 'Parallax'
  2017 = 'PARK CASSEGRAIN'
  2090 = 'Park telescope'
  2091 = 'Park telescope ...'
  2085 = 'Park the telescope at:'
  1213 = 'Pattern length (no. of bits of the pattern to use)'
  1495 = 'Peak current'
  119 = 'Peak current limit'
  1811 = 'Permanent brake control:'
  1250 = 'Person entered dome'
  1985 = 'Person entered dome, \npower is OFF'
  1984 = 'Person entered dome, power is OFF'
  1219 = 'Person has entered'
  1243 = 'Person has entered  without bypass'
  1993 = 'Person has entered dome'
  1253 = 'Person has entered the dome'
  1185 = 'Person has entered the dome area'
  1244 = 'Person has entered without bypass'
  1220 = 'Person has left'
  1248 = 'Person safety'
  1249 = 'Person safety OK'
  1247 = 'PG: Pumps Group box'
  1632 = 'Physical axis'
  641 = 'Pneumatic \nsupply \npressure'
  642 = 'Pneumatic \nsupply pressure'
  640 = 'Pneumatic supply\npressure'
  573 = 'Pneumatic supply \nsensor alarms\n[bar]'
  569 = 'Pneumatic supply \nsensor alarms:'
  639 = 'Pneumatic supply pressure'
  568 = 'Pneumatic supply sensor alarms:'
  566 = 'Pneumatic supply sensor full scale [bar]'
  1766 = 'Point'
  1438 = 'Point axes'
  1433 = 'Point telescope'
  1778 = 'Point telescope ...'
  1777 = 'Point the telescope'
  1439 = 'Pointing'
  2077 = 'Pointing and tracking'
  2081 = 'Pointing model active'
  2056 = 'Pointing model active:'
  1382 = 'Pointing status (by C++ task)'
  1348 = 'Polar motion '
  180 = 'Polarity'
  170 = 'Port'
  408 = 'Port status'
  153 = 'POS DRIVE'
  94 = 'Pos. axis'
  124 = 'Pos. ctrl. Integral term'
  123 = 'Pos. ctrl. Proport. term'
  227 = 'Pos. motor actual current'
  229 = 'POS. motor actual current'
  230 = 'POS. motor average current'
  438 = 'PosDiff %.2f°'
  97 = 'Positiioning\naxis'
  95 = 'Positiioning axis'
  96 = 'Positiioningaxis'
  126 = 'Position'
  1047 = 'Position\nmeasurement'
  442 = 'Position %.2f°'
  87 = 'Position difference'
  79 = 'Position error'
  410 = 'Position fix'
  1046 = 'Position measurement'
  2101 = 'Position on sky'
  1684 = 'Position setpoint generator'
  249 = 'Positioning\n(ABL)'
  250 = 'Positioning\n(POS)'
  90 = 'Positioning\naxis'
  98 = 'Positioning\ndrive'
  154 = 'POSITIONING\nDRIVE'
  251 = 'Positioning motor\n(POS)'
  225 = 'Positioning motor actual current'
  1072 = 'Positioning procedure'
  89 = 'Positioningaxis'
  1598 = 'Positions'
  1641 = 'Positive'
  183 = 'Positive Limit Switch'
  265 = 'Positive limit [mm]'
  215 = 'Positive soft limit'
  263 = 'Positive soft limit [mm]'
  301 = 'Positive soft limit [°]'
  1511 = 'Positive torque limit'
  15 = 'Power'
  439 = 'power'
  756 = 'Power off'
  1804 = 'Power OFF'
  2023 = 'Power off ROC'
  2022 = 'Power off ROC (if it was powered on)'
  2025 = 'Power off the Cassegrain rotator (ROC)'
  2027 = 'Power off the Cassegrain rotator (RON)'
  757 = 'Power on'
  1803 = 'Power ON'
  755 = 'Power on for %d seconds'
  2021 = 'Power on ROC'
  2024 = 'Power on the Cassegrain rotator (ROC)'
  2026 = 'Power on the Cassegrain rotator (RON)'
  754 = 'Power relay'
  440 = 'powered'
  1640 = 'Powered'
  1983 = 'Powered off \n(person entered dome)'
  1982 = 'Powered off (person \nentered dome)'
  1981 = 'Powered off (person entered dome)'
  1987 = 'Powered off due \nto person entering dome'
  1988 = 'Powered off due to\nperson entering dome'
  1986 = 'Powered off due to person'
  1636 = 'POX'
  1637 = 'POY'
  2094 = 'Prefer direction with most travel left instead of shortest path'
  2053 = 'Prefer most travel left'
  681 = 'Press the buttons in ascending order to login'
  680 = 'Press the buttons in ascending order to unlock the screen'
  679 = 'Press the buttons in the correct order to unlock the screen'
  576 = 'Pressure @ mirror cell\nalarms [bar]'
  637 = 'Pressure @ mirror cell\n[bar]'
  575 = 'Pressure @ mirror cell sensor full scale [bar]'
  636 = 'Pressure @ mirror cell [bar]'
  635 = 'Pressure @ mirror cell[bar]'
  574 = 'Pressure @ regulator\nalarms [bar]'
  572 = 'Pressure @ regulator\nalarms:'
  638 = 'Pressure @ regulator\n[bar]'
  571 = 'Pressure @ regulator alarms:'
  570 = 'Pressure @ regulator sensor full scale [bar]'
  1003 = 'Pressure measurement [Bar]'
  1002 = 'Pressure measurement [°C]'
  607 = 'Pressure regulator range [bar]'
  860 = 'Pressure rises\nduring startup\n(QMin -> 0)'
  861 = 'Pressure rises\nduring startup\n(Underpressure -> 0)'
  925 = 'Pressure rising'
  928 = 'Pressure rising after startup'
  927 = 'Pressure rising at startup'
  865 = 'Pressure rising error'
  863 = 'Pressure rising error\nduring startup\n(Underpressure -> 0)'
  999 = 'Pressure sensor full scale'
  1000 = 'Pressure sensor full scale [Bar]'
  539 = 'Pressure setpoint'
  1536 = 'Primary operation mode'
  982 = 'Procedure status:'
  1078 = 'Procedures'
  978 = 'Pumps enabled'
  911 = 'Pumps not starting'
  909 = 'Pumps not starting up'
  894 = 'Pumps not stopped'
  912 = 'Pumps not stopping'
  1335 = 'Pumps power OK'
  1336 = 'Pumps powered'
  892 = 'Pumps release'
  895 = 'Pumps release \n(RFR ReglerFreigabe)'
  1016 = 'Pumps released'
  953 = 'Pumps running'
  873 = 'Pumps starting'
  983 = 'Pumps starting and stopping'
  910 = 'Pumps starting up'
  831 = 'Pumps startup'
  979 = 'Pumps state'
  1014 = 'Pumps status'
  871 = 'Pumps stopped'
  872 = 'Pumps stopped detection'
  869 = 'Pumps stopping'
  1313 = 'Put the X, Y, Tilt X and Tilt Y axes at their default initial positions'
  1311 = 'Put the X, Y, Tilt X and Tilt Y axes at their default positions'
  1309 = 'Put the X, Y, Tilt X and Tilt Y axes at their fixed positions'
  1401 = 'Quick calculations'
  1969 = 'Quick stop'
  1970 = 'Quick stop deceleration'
  1971 = 'Quick stop jerk'
  1972 = 'QuickStop axes'
  206 = 'R'
  1615 = 'R.A.'
  1371 = 'rad'
  1440 = 'Rad'
  1374 = 'rad/year'
  623 = 'Radia; pressure\n@ regulator'
  615 = 'Radial pressure'
  616 = 'Radial pressure\n@ mirror cell'
  624 = 'Radial pressure\n@ regulator'
  629 = 'Radial regulator\nsetpoint'
  562 = 'Radial support'
  565 = 'Radial support setpoint selection'
  563 = 'Radial support status'
  645 = 'Radial support vacuum'
  1377 = 'Radial velocity'
  578 = 'RadialPressureSetpoint = CorrectionCoefficient * 1.33 bar * cos(elevation)'
  1441 = 'Radians'
  1497 = 'Rated current'
  684 = 'Re-\ninitialize'
  107 = 'Read'
  969 = 'REBOOT'
  683 = 'Reinitialize'
  517 = 'Relative humidities'
  1362 = 'Relative humidity, fixed by config [degrees]'
  1365 = 'Relative humidity, fixed by config [fraction, 0..1]'
  459 = 'Relay'
  464 = 'Relay (all 4 magnets!)'
  460 = 'Relay (all 4 panels!)'
  1152 = 'Relay 1 is closed'
  25 = 'Reset'
  202 = 'Reset\nerror(s)'
  1036 = 'Reset bottom'
  1038 = 'Reset bottom drive'
  512 = 'Reset error(s)'
  436 = 'Reset errors'
  822 = 'Reset hydraulics errors'
  820 = 'Reset hydraulics safety'
  1432 = 'Reset temporary safety'
  1034 = 'Reset the drives'
  1937 = 'Reset to zero'
  1035 = 'Reset top'
  1037 = 'Reset top drive'
  86 = 'Residual'
  773 = 'Restart'
  1416 = 'Restart & \ntroubleshoot'
  800 = 'Restart emergency stops'
  774 = 'Restart hydraulics safety'
  905 = 'Restart hydraulics safety\n(this expects '
  821 = 'Restart pumps'
  110 = 'Result'
  108 = 'Result:'
  109 = 'Result: value'
  973 = 'return'
  974 = 'Return\nfilter'
  1184 = 'Return button is being pushed'
  1150 = 'Return button is pushed'
  829 = 'Return filter'
  889 = 'Return filter OK'
  1395 = 'Reverse calculations'
  1396 = 'Right Ascention'
  2099 = 'RMS error'
  1522 = 'RMS error (1 sec)'
  1517 = 'RMS error 1 sec'
  1649 = 'ROC'
  1782 = 'roc'
  2071 = 'ROC position angle (sky rotation) sign (-1 is negative, 1 is positive)'
  2069 = 'ROC position angle sign (-1 is negative, 1 is positive)'
  2009 = 'ROC position to go to, in degrees'
  1650 = 'RON'
  1783 = 'ron'
  2072 = 'RON position angle (sky rotation) sign (-1 is negative, 1 is positive)'
  2070 = 'RON position angle sign (-1 is negative, 1 is positive)'
  1617 = 'rot'
  1755 = 'Rot'
  236 = 'ROT motor position'
  2011 = 'ROT position to go to, in degrees'
  1848 = 'Rot. Cas.'
  74 = 'ROTATION'
  76 = 'Rotation'
  1620 = 'rotation'
  130 = 'Rotation\nABL drive'
  128 = 'Rotation\ndrive'
  131 = 'Rotation\nPOS drive'
  129 = 'Rotation\npos. drive'
  1239 = 'Rotation axes release'
  1238 = 'Rotation axis release'
  1849 = 'Rotation Cas.'
  139 = 'Rotation offset [°]'
  138 = 'Rotation position [°]'
  203 = 'Rotation status'
  1850 = 'Rotator Cas.'
  1847 = 'Rotator Cassegrain'
  1852 = 'Rotator Nas.'
  1851 = 'Rotator Nasm.'
  2034 = 'Rotator(s)'
  294 = 'RxError counter'
  295 = 'RxError counter:'
  80 = 's'
  1561 = 'S\n180°'
  1558 = 'S 180°'
  1994 = 'Safe access'
  1122 = 'Safe to enter'
  1124 = 'safe to enter'
  2106 = 'Safety'
  897 = 'Safety group'
  811 = 'Safety group errors'
  810 = 'Safety group errprs'
  824 = 'Safety logic'
  6 = 'SAVE'
  1710 = 'Scale the ABL output torque by this fraction value (only for testing purposes, must be 1 normally!)'
  1711 = 'Scale the ABL torque by this fraction (only for testing purposes, must be 1 normally!)'
  100 = 'SDO read'
  174 = 'SDO write'
  1807 = 'sec'
  759 = 'Seconds remaining: %.1f'
  758 = 'Seconds remaining: %d'
  1322 = 'Selec newt instrument'
  325 = 'Select focal station:'
  1321 = 'Select instrument'
  1090 = 'Select instrument ...'
  326 = 'Select new focal station for M3:'
  1323 = 'Select new instrument'
  469 = 'Selected Panel'
  474 = 'Selected panel'
  175 = 'Send at initialization'
  118 = 'Send initially'
  1033 = 'Send start command to safety'
  1109 = 'Sensor 1'
  1108 = 'Sensor 1 +X'
  1110 = 'Sensor 2'
  1174 = 'Sensors are being bypassed'
  1173 = 'Sensors are bypassed permanently'
  404 = 'Serial communication checksum status'
  399 = 'Serial communication data status'
  398 = 'Serial communication link receiving'
  397 = 'Serial communication link status'
  400 = 'Serial communication port status'
  406 = 'Serial communication status'
  401 = 'Serial communication transmission status'
  333 = 'Service'
  1878 = 'Set a velocity in alpha / delta'
  548 = 'Set AUTO'
  555 = 'Set automatic'
  1539 = 'Set brake state'
  1574 = 'Set counter done'
  414 = 'Set manual'
  1381 = 'Set new target'
  2107 = 'Set position'
  1368 = 'Set target'
  1765 = 'Set target ...'
  2029 = 'Set the cassegrain rotator (ROC) as active'
  2030 = 'Set the cassegrain rotator (ROC) as active (ROT)'
  2031 = 'Set the cassegrain rotator (ROC) as active (so ROT = ROC)'
  2032 = 'Set the nasmyth rotator (RON) as active (so RON = ROC)'
  2033 = 'Set the nasmyth rotator (RON) as active (so ROT = RON)'
  1314 = 'Set the X, Y, Tilt X and Tilt Y axes at their default initial positions'
  1921 = 'Set velocity\nalpha / delta'
  1919 = 'Set velocity in\nalpha / delta'
  544 = 'Setpoint'
  1606 = 'Setpoint\ngenerator'
  1605 = 'Setpoint generator'
  1824 = 'SetPos'
  1943 = 'SetVelo'
  1482 = 'Show parameters'
  2012 = 'Show position:'
  11 = 'Shut down'
  970 = 'Shutdown\n(TECH only)'
  1013 = 'SIMULATION ACTIVE'
  1607 = 'Slalib'
  1146 = 'Sleeping'
  1695 = 'Slip monitoring: maximum difference between motor encoders and LIDAs, in degrees'
  1691 = 'Slit limit: maximum difference between motor encorders and LIDAs'
  1692 = 'Slit limit: maximum difference between motor encorders and LIDAs, in degrees'
  1694 = 'Slit monitoring: maximum difference between motor encoders and LIDAs, in degrees'
  1693 = 'Slit monitoring: maximum difference between motor encorders and LIDAs, in degrees'
  1730 = 'SLOW'
  613 = 'SO'
  534 = 'SO\n'
  535 = 'SO\n '
  1659 = 'Software limits'
  1660 = 'Software position limits'
  597 = 'South sensor alarms [daN]'
  598 = 'South sensor alarms [daN]\n(SO)'
  596 = 'South sensor alarms[daN]'
  632 = 'South sensor [daN]\n(SO)'
  1048 = 'SSI encoder'
  1421 = 'Staff only'
  1175 = 'STAFF ONLY: sensor bypassing'
  266 = 'Standstill tolerance [mm/s]'
  151 = 'Standstill tolerance [°/s]'
  1328 = 'START'
  1614 = 'start'
  239 = 'Start calibration'
  1327 = 'Start changing the instrument'
  273 = 'Start homing'
  1436 = 'Start tracking after pointing'
  1776 = 'Start tracking the new target'
  980 = 'Start up pumps'
  830 = 'Starting up'
  828 = 'Startup command'
  907 = 'Startup pulse'
  908 = 'Startup pulse 0 -> 1 -> 0'
  906 = 'Startup trigger'
  2105 = 'Statistics'
  542 = 'Status'
  1604 = 'Status inp.'
  1585 = 'Status of:'
  932 = 'Statuses'
  1932 = 'step'
  761 = 'Steps'
  1067 = 'Steps around final position to go to first'
  1066 = 'Steps before final position'
  1304 = 'Steps between final and anti-backlash position'
  1305 = 'Steps between final and close position'
  1069 = 'Steps between final and one-but-final position'
  1068 = 'Steps for the one-but-final move'
  768 = 'Steps remaining: %d'
  1324 = 'Steps to be executed'
  93 = 'STOP'
  201 = 'Stop'
  1793 = 'STOP\nALL'
  1801 = 'STOP\nAZI'
  1949 = 'STOP\nazimuth'
  1950 = 'STOP\nBOTH'
  1800 = 'STOP\nELE'
  1951 = 'STOP\nelevation'
  2093 = 'STOP\nmoving'
  1802 = 'STOP\nROC'
  2092 = 'STOP\ntelescope'
  2114 = 'STOP\ntracking / moving'
  2115 = 'STOP\ntracking, moving, ...'
  92 = 'Stop all motion'
  1445 = 'Stop axes'
  1177 = 'Stop bypassing'
  1948 = 'Stop individual axes'
  981 = 'Stop pumps'
  2075 = 'Stop telescope'
  1602 = 'Sts input'
  102 = 'SubIndex'
  1965 = 'Sufficiently high'
  1968 = 'Sufficiently high to calculate refraction'
  1599 = 'Summary'
  549 = 'Switch to AUTO'
  558 = 'Switch to automatic'
  559 = 'Switch to fixed'
  550 = 'Switch to MANUAL'
  1052 = 'Sync'
  1584 = 'Sync error'
  444 = 'System'
  207 = 'T'
  724 = 't'
  955 = 'T\nO\nP'
  342 = 'TAI to UTC (no. of leap seconds)'
  196 = 'Target'
  416 = 'Target distance between panels [°]'
  508 = 'Target for rotation:'
  509 = 'Target for translation:'
  210 = 'Target mirror position'
  212 = 'Target motor offset'
  82 = 'Target offset'
  16 = 'Target position'
  241 = 'Target velocity'
  1825 = 'TargetPos'
  31 = 'Tech'
  662 = 'TECH'
  514 = 'TELEMETRY'
  674 = 'Telemetry'
  1254 = 'Telescope'
  1412 = 'TELESCOPE'
  1199 = 'Telescope\nunblocked'
  916 = 'Telescope axes release'
  915 = 'Telescope Azimuth axis release'
  1121 = 'Telescope blocked'
  1120 = 'Telescope blocked\nsafe'
  1123 = 'Telescope blocked,'
  1125 = 'Telescope blocked,\nsafe to enter'
  1138 = 'Telescope is unblocked permanently'
  1142 = 'Telescope status'
  1198 = 'Telescope unblocked'
  1408 = 'TELESOCPE'
  516 = 'Temperatures'
  1257 = 'Test'
  1464 = 'TF'
  1699 = 'The ABL torque can fall maximum ... Nm/s on the telescope axis (always >0)'
  1698 = 'The ABL torque can rise maximum ... Nm/s on the telescope axis (always >0)'
  1708 = 'The ABL torque when the axis is not accelerating or decelerating (always >0)'
  1709 = 'The ABL torque when the AZI axis is not accelerating or decelerating (always >0)'
  1704 = 'The maximum ABL torque (acceleration > 0) in Nm/s on the telescope axis (always >0)'
  1706 = 'The maximum ABL torque (AZI acceleration > 0) in Nm/s on the telescope axis (always >0)'
  1702 = 'The maximum ABL torque (during acceleration) in Nm/s on the telescope axis (always >0)'
  1700 = 'The maximum ABL torque in Nm/s on the telescope axis (always >0)'
  1722 = 'The maximum acceleration setpoint of the axis in degrees/sec^2'
  1689 = 'The maximum bidirectional velocity setpoint of the axis in degrees/sec (>0)'
  1687 = 'The maximum position setpoint of the axis in degrees (a bit before the soft limit)'
  1690 = 'The maximum velocity setpoint (bidirectional) of the axis in degrees/sec (>0)'
  1688 = 'The maximum velocity setpoint of the axis in degrees/sec'
  1705 = 'The minimum ABL torque (acceleration < 0) in Nm/s on the telescope axis (always >0)'
  1707 = 'The minimum ABL torque (AZI acceleration < 0) in Nm/s on the telescope axis (always >0)'
  1703 = 'The minimum ABL torque (during deceleration) in Nm/s on the telescope axis (always >0)'
  1701 = 'The minimum ABL torque in Nm/s on the telescope axis (always >0)'
  1685 = 'The minimum position setpoint of the axis in degrees'
  1686 = 'The minimum position setpoint of the axis in degrees (a bit before the soft limit)'
  730 = 'The number of steps to be expected between the time at which the PLC realizes that the brake signal must be set, and the time that the axis is fully stopped (for Z axis: at low speed)'
  732 = 'The number of steps which should be carried out at minimum to counter-act the backlash in the system during the final move (for Z axis: at low speed)'
  1828 = 'The position of the homing mark (in degrees), with respect to the absolute zero'
  1829 = 'The position of the homing mark (in degrees), with respect to the absolute zero azimuth'
  1638 = 'The x-coordinate of a pointing origin on a derotator'
  1639 = 'The y-coordinate of a pointing origin on a derotator'
  687 = 'The Z axis'
  965 = 'Then, double-click the "Mercator TCS GUI" icon,\nand wait a few seconds for the GUI to show up.'
  966 = 'Then, double-click the "Mercator TCS GUI" icon, \nand wait a few seconds \nfor the GUI to show up.'
  967 = 'Then, double-click the "Mercator TCS GUI" icon, and wait a few seconds \nfor the GUI to show up.'
  1080 = 'Thermal focus'
  1092 = 'Thermal focus for all focal stations'
  1095 = 'Thermal focus for all focal stations:'
  1081 = 'Thermal focus for current instrument'
  1091 = 'Thermal focus for other focal stations'
  1307 = 'Thermal focus for other focal stations:'
  1084 = 'Thermal focus of Z axis'
  703 = 'thermalFocusZ  =  offset + t * topTemperature'
  704 = 'thermalFocusZ  =  offset + t * topTemperature + c * centreTemperature + m * mirrorCellTemperature'
  706 = 'thermalFocusZ  =  offset + top * topTemperature + c * centreTemperature + m * mirrorCellTemperature'
  707 = 'thermalFocusZ  =  offset + top * topTemperature + centre * centreTemperature + m * mirrorCellTemperature'
  708 = 'thermalFocusZ  =  offset + top * topTemperature + centre * centreTemperature + mirrorCell * mirrorCellTemperature'
  723 = 'thermalFocusZ [mm] =  o'
  714 = 'thermalFocusZ [mm] =  offset'
  712 = 'thermalFocusZ [mm] =  offset + top * topTemperature + centre * centreTemperature + mirrorCell * mirrorCellTemperature'
  1054 = 'Tilt X'
  1289 = 'Tilt X fixed position tolerance [mm]'
  1288 = 'Tilt X fixed position [mm]'
  1061 = 'Tilt Y'
  1291 = 'Tilt Y fixed position tolerance [mm]'
  1290 = 'Tilt Y fixed position [mm]'
  368 = 'Time'
  1399 = 'Time & Hour Angle'
  733 = 'Time (in seconds) to wait after the axis has been moved'
